# B&R Automation Studio project Panasonic_LinkaKapacitorov_A2021040 (part 4)

#### Main.st - Init, cyclic, exit code
```iecst
PROGRAM _INIT
	(* Insert code here *)

END_PROGRAM

PROGRAM _CYCLIC

	//Volanie podprogramov//
	OvlCentrovacky;
	OvlCitackyRFID;
	OvlTlaciarne;

	//Volanie funkcie SequenceControl//
	SequenceControl(SC:= SC_StoperEtiketovania);

	//Volanie funkčného bloku komunikácie Panasonic//
	KOM_Panasonic();

	//Reset sekcie //
	IF StoperEtiketovania.Reset THEN
		SC_StoperEtiketovania.Step:= 0;
		StoperEtiketovania.Reset:= FALSE;
	ELSIF NOT Safety.STAV.ZonaCS_AKTIVNA THEN
		SC_StoperEtiketovania.Step:= 0;
	END_IF

	//Status Tlačiareň zaaretovaná//
	StoperEtiketovania.STAV.TlaciarenZaaretovana:= StoperEtiketovania.IN.SuflikTlaciarne_LS_IS23 AND StoperEtiketovania.IN.SuflikTlaciarne_PS_IS22;

	//Zrušenie príznaku prebieha vyvezenie paletky//
	IF StoperEtiketovania.STAV.PrebiehaVyvazaniePaletky AND StoperDopravNG.IN.Stoper_PritomnostPaletky_IS15 THEN
		StoperEtiketovania.STAV.PrebiehaVyvazaniePaletky:= FALSE;
	END_IF

	//Označenie paletky NG pri otvoreni dverí//
	IF NOT Safety.STAV.ZamkyBunky_AKTIVNE AND RFID_Hlava_2.STAV.PritomnostCipu AND RFID_Hlava_2.PAR.PrecitaneCisloPaletky <> '' THEN
		i:=  STRING_TO_USINT(RFID_Hlava_2.PAR.PrecitaneCisloPaletky);
		IF NOT Paletka[i].StavKomunikacie_DONE THEN
			Paletka[i].StavPaletky:= 'NG';
		END_IF
	END_IF

	CASE SC_StoperEtiketovania.Step OF

		0:
			SC_StoperEtiketovania.StepName:='0 - Nulovanie';
			StoperEtiketovania.Automat:= FALSE;
			StoperEtiketovania.KoniecCyklu:= FALSE;
			StoperEtiketovania.Manual:= FALSE;
			StoperEtiketovania.STAV.PoINIT:= FALSE;
			StoperEtiketovania.OUT.StoperZASUN_YV007:= FALSE;
			SC_OvlCentrovacky.Step:= 0;
			Robot.KOM_OUT.PresunDoPozicieOdobratiaEtikety:= FALSE;
			Robot.KOM_OUT.PresunDoMutingPozicie:= FALSE;
			Robot.KOM_OUT.PresunDoPoziceKontrolyEtikety:= FALSE;
			Robot.KOM_OUT.PresunDoPoziceKontrEtiketyPriamo:= FALSE;
			Robot.KOM_OUT.PresunDoPozicieKontrolyIntStitku:= FALSE;
			Robot.KOM_OUT.NalepEtiketu:= FALSE;
			Robot.KOM_OUT.CitanieStitkuUkoncene:= FALSE;
			StoperEtiketovania.OUT.Tlaciaren_VytlacEtiketu:= FALSE;
			StoperEtiketovania.OUT.Tlaciaren_VytlacZnovaEtiketu:= FALSE;
			Kamera.STAV.Results_READY:= FALSE;
			Kamera.CMD.Triger:= FALSE;
			StoperEtiketovania.STAV.PrebiehaVyvazaniePaletky:= FALSE;
			StoperEtiketovania.RR_VytlacEtiketu:= FALSE;
			Vizu.ZobrazHlasenie_ZaaretujTlaciaren:= 1;
			Vizu.ZobrazHlas_ZatvorSerDvereTlac:= 1;
			Vizu.ZobrazHlasenie_TlaciarenOffline:= 1;
			StoperDopravNG.OUT.NatlakujTlmicPaletky_YV008:= FALSE;
			NacitanieKorekcii_DONE:= FALSE;
			StoperEtiketovania.STAV.Etiketovanie_BUSY:= FALSE;
			StoperEtiketovania_Statistika.IN.START_MeraniaCasu:= FALSE;
			KOM_Panasonic.Server_IN.DataForServer_READY:= FALSE;
			KOM_Panasonic.Server_IN.VytlacEtiketu_RucnyRezim:= FALSE;
			KOM_Panasonic.Server_IN.ProcessResult:= FALSE;
			KOM_Panasonic.Server_IN.Blowing_Error:= FALSE;
			KOM_Panasonic.Server_IN.DMcode_Reading_Error:= FALSE;
			KOM_Panasonic.Server_IN.QRcode_Reading_Error:= FALSE;
			KOM_Panasonic.Server_IN.RFID_Reading_Error:= FALSE;
			KOM_Panasonic.Server_IN.Text_Reading_Error:= FALSE;
			KOM_Panasonic.Server_IN.CommandNumber:= 0;
			KOM_Panasonic.Server_IN.RezimBezTlaceEtikety:= FALSE;
			StoperEtiketovania.STAV.Warning:= FALSE;

			IF Safety.STAV.ZonaCS_AKTIVNA AND Safety.STAV.ZonaBunky_AKTIVNA AND Linka.IN.TlakVzduchu_OK_S2 AND NOT NastalaPorucha AND Linka.STAV.Hardware_OK THEN
				SC_StoperEtiketovania.ResetStep:= TRUE;
				SC_StoperEtiketovania.Step:= 1;
			END_IF

		1:
			SC_StoperEtiketovania.StepName:='1 - Cakam na spustenie vyroby';
			StoperEtiketovania.KoniecCyklu:= FALSE;
			IF StoperEtiketovania.Automat THEN
				SC_StoperEtiketovania.Step:= 2;
			ELSIF StoperEtiketovania.Manual THEN
				SC_StoperEtiketovania.Step:= 700;
			END_IF

			//********************************************************Inicializácia****************************************************************************//

		2:
			SC_StoperEtiketovania.StepName:='2 - Inicializacia - cakam na spustenie inicializacie';
			SC_StoperEtiketovania.IdleTime.PT:= T#4s;
			SC_StoperEtiketovania.AlarmTime.PT:= T#5s;

			IF DopravBunky.STAV.PoINIT AND Robot.STAV.PoINIT THEN
				SC_StoperEtiketovania.ResetStep:= TRUE;
				SC_StoperEtiketovania.Step:= 10;
			END_IF

		10:
			SC_StoperEtiketovania.StepName:='10 - Inicializacia - zasunutie centrovacky';
			SC_StoperEtiketovania.IdleTime.PT:= T#4s;
			SC_StoperEtiketovania.AlarmTime.PT:= T#5s;

			IF NOT SC_StoperEtiketovania.Switch1 THEN
				Centrovacku_ZASUN:= TRUE;
				SC_StoperEtiketovania.Switch1:= TRUE;
			END_IF

			IF StoperEtiketovania.IN.Centrovanie_SpodnaPoloha_IS17 THEN
				SC_StoperEtiketovania.ResetStep:= TRUE;
				SC_StoperEtiketovania.Step:= 13;
			END_IF

		13:
			SC_StoperEtiketovania.StepName:='13 - Inicializacia - hladanie paletky';
			SC_StoperEtiketovania.IdleTime.PT:= T#5s;
			SC_StoperEtiketovania.AlarmTime.PT:= T#5s;
			SC_StoperEtiketovania.IdleTime.IN:= TRUE;

			IF StoperEtiketovania.IN.PritomnostPaletky_IS16 THEN
				StoperEtiketovania.STAV.PoINIT:= TRUE;
				SC_StoperEtiketovania.ResetStep:= TRUE;
				SC_StoperEtiketovania.Step:= 100;
			ELSIF SC_StoperEtiketovania.IdleTime.Q THEN
				StoperEtiketovania.STAV.PoINIT:= TRUE;
				SC_StoperEtiketovania.ResetStep:= TRUE;
				SC_StoperEtiketovania.Step:= 100;
			END_IF

			//********************************************************Automatický režim****************************************************************************//
		100:
			SC_StoperEtiketovania.StepName:='100 - Automaticky Rezim - cakam na príchod paletky na stoper';
			SC_StoperEtiketovania.IdleTime.PT:= T#200ms;
			SC_StoperEtiketovania.AlarmTime.PT:= T#5s;

			IF Linka.Rezim_BezTlaceEtikety THEN
				KOM_Panasonic.Server_IN.RezimBezTlaceEtikety:= TRUE;
			ELSE
				KOM_Panasonic.Server_IN.RezimBezTlaceEtikety:= FALSE;
			END_IF

			SC_StoperEtiketovania.IdleTime.IN:= StoperEtiketovania.IN.PritomnostPaletky_IS16;

			IF StoperEtiketovania.KoniecCyklu THEN
				SC_StoperEtiketovania.ResetStep:= TRUE;
				SC_StoperEtiketovania.Step:= 0;
			ELSIF SC_StoperEtiketovania.IdleTime.Q THEN
				StoperEtiketovania_Statistika.IN.START_MeraniaCasu:= TRUE;
				StoperEtiketovania_Statistika.IN.ZAPIS_MeraniaCasu:= TRUE;
				SC_StoperEtiketovania.ResetStep:= TRUE;
				SC_StoperEtiketovania.Step:= 103;
			END_IF

		103:
			SC_StoperEtiketovania.StepName:='103 - Automaticky Rezim - citam cislo paletky';
			SC_StoperEtiketovania.IdleTime.PT:= T#0ms;
			SC_StoperEtiketovania.AlarmTime.PT:= T#10s;

			SC_StoperEtiketovania.IdleTime.IN:= RFID_Hlava_2.STAV.PritomnostCipu;

			IF SC_StoperEtiketovania.IdleTime.Q THEN
				IF RFID_Hlava_2.PAR.PrecitaneCisloPaletky <> '' THEN
					i:=  STRING_TO_USINT(RFID_Hlava_2.PAR.PrecitaneCisloPaletky);
					IF Linka.Rezim_Priechodny THEN
						SC_StoperEtiketovania.ResetStep:= TRUE;
						SC_StoperEtiketovania.Step:= 240;
					ELSE
						SC_StoperEtiketovania.ResetStep:= TRUE;
						SC_StoperEtiketovania.Step:= 105;
					END_IF
				ELSE
					Alarmy[61]:= TRUE;
					PoruchaBunky:= TRUE;
					SC_StoperEtiketovania.ResetStep:= TRUE;
					SC_StoperEtiketovania.Step:= 0;
				END_IF
			END_IF

		105:
			SC_StoperEtiketovania.StepName:='108 - Automaticky Rezim - nacitanie offsetov pozicie lepenia zakaznickej etikety a cisla programu pre robot';
			SC_StoperEtiketovania.IdleTime.PT:= T#200ms;
			SC_StoperEtiketovania.AlarmTime.PT:= T#10s;

			OffsetRobota_NazovModelu:= Paletka[i].NazovModelu;
			Robot.KOM_OUT.CisloProduktu:= Paletka[i].Robot_CisloProgramu;
			IF Kamera.STAV.AktualneCisloProgramu <> Paletka[i].Kamera_CisloProgramu_QRkod THEN
				Kamera.PAR.ZadaneCisloProgramu:= Paletka[i].Kamera_CisloProgramu_QRkod;
			END_IF

			IF NOT SC_StoperEtiketovania.Switch1 THEN
				NacitajKorekcieRobota:= TRUE;
				SC_StoperEtiketovania.Switch1:= TRUE;
			END_IF

			IF NacitanieKorekcii_DONE THEN
				NacitanieKorekcii_DONE:= FALSE;
				IF Linka.PAR.Zvolena_PozLepenia_OffsetX <> 0 THEN
					IF Linka.PAR.Zvolena_PozLepenia_OffsetX > 0 THEN
						Robot.KOM_OUT.LepenieStitku_OffsetX:= REAL_TO_USINT(Linka.PAR.Zvolena_PozLepenia_OffsetX * 10);
						Robot.KOM_OUT.LepenieStitku_ZnamienkoOffsetX:= FALSE;
					ELSIF Linka.PAR.Zvolena_PozLepenia_OffsetX < 0 THEN
						Robot.KOM_OUT.LepenieStitku_OffsetX:= REAL_TO_USINT(ABS(Linka.PAR.Zvolena_PozLepenia_OffsetX) * 10);
						Robot.KOM_OUT.LepenieStitku_ZnamienkoOffsetX:= TRUE;
					END_IF
				ELSE
					Robot.KOM_OUT.LepenieStitku_OffsetX:= 0;
					Robot.KOM_OUT.LepenieStitku_ZnamienkoOffsetX:= FALSE;
				END_IF
				IF Linka.PAR.Zvolena_PozLepenia_OffsetY <> 0 THEN
					IF Linka.PAR.Zvolena_PozLepenia_OffsetY > 0 THEN
						Robot.KOM_OUT.LepenieStitku_OffsetY:= REAL_TO_USINT(Linka.PAR.Zvolena_PozLepenia_OffsetY * 10);
						Robot.KOM_OUT.LepenieStitku_ZnamienkoOffsetY:= FALSE;
					ELSIF Linka.PAR.Zvolena_PozLepenia_OffsetY < 0 THEN
						Robot.KOM_OUT.LepenieStitku_OffsetY:= REAL_TO_USINT(ABS(Linka.PAR.Zvolena_PozLepenia_OffsetY) * 10);
						Robot.KOM_OUT.LepenieStitku_ZnamienkoOffsetY:= TRUE;
					END_IF
				ELSE
					Robot.KOM_OUT.LepenieStitku_OffsetY:= 0;
					Robot.KOM_OUT.LepenieStitku_ZnamienkoOffsetY:= FALSE;
				END_IF
				IF Linka.PAR.Zvolena_PozLepenia_OffsetZ <> 0 THEN
					IF Linka.PAR.Zvolena_PozLepenia_OffsetZ > 0 THEN
						Robot.KOM_OUT.LepenieStitku_OffsetZ:= REAL_TO_USINT(Linka.PAR.Zvolena_PozLepenia_OffsetZ * 10);
						Robot.KOM_OUT.LepenieStitku_ZnamienkoOffsetZ:= FALSE;
					ELSIF Linka.PAR.Zvolena_PozLepenia_OffsetZ < 0 THEN
						Robot.KOM_OUT.LepenieStitku_OffsetZ:= REAL_TO_USINT(ABS(Linka.PAR.Zvolena_PozLepenia_OffsetZ) * 10);
						Robot.KOM_OUT.LepenieStitku_ZnamienkoOffsetZ:= TRUE;
					END_IF
				ELSE
					Robot.KOM_OUT.LepenieStitku_OffsetZ:= 0;
					Robot.KOM_OUT.LepenieStitku_ZnamienkoOffsetZ:= FALSE;
				END_IF
				SC_StoperEtiketovania.ResetStep:= TRUE;
				SC_StoperEtiketovania.Step:= 110;
			END_IF

		110:
			SC_StoperEtiketovania.StepName:='110 - Automaticky Rezim - zacentrovanie paletky';
			SC_StoperEtiketovania.IdleTime.PT:= T#200ms;
			SC_StoperEtiketovania.AlarmTime.PT:= T#5s;

			IF NOT SC_StoperEtiketovania.Switch1 THEN
				Centrovacku_VYSUN:= TRUE;
				SC_StoperEtiketovania.Switch1:= TRUE;
			END_IF

			IF StoperEtiketovania.IN.Centrovanie_HornaPoloha_IS18 AND NOT StoperDopravNG.STAV.DopravnikNG_BUSY THEN
				IF Linka.Rezim_BezKomunikacie THEN
					SC_StoperEtiketovania.ResetStep:= TRUE;
					SC_StoperEtiketovania.Step:= 115;
				ELSE
					SC_StoperEtiketovania.ResetStep:= TRUE;
					SC_StoperEtiketovania.Step:= 113;
				END_IF
			END_IF

		113:
			SC_StoperEtiketovania.StepName:='113 - Automaticky Rezim - kontrola stavu komunikacie a paletky';
			SC_StoperEtiketovania.IdleTime.PT:= T#200ms;
			SC_StoperEtiketovania.AlarmTime.PT:= T#5s;

			IF Paletka[i].StavKomunikacie_DONE THEN
				SC_StoperEtiketovania.ResetStep:= TRUE;
				SC_StoperEtiketovania.Step:= 240;
			ELSIF Paletka[i].StavPaletky = 'PR' THEN	//Priechodný režim
				SC_StoperEtiketovania.ResetStep:= TRUE;
				SC_StoperEtiketovania.Step:= 240;
			ELSIF Paletka[i].StavPaletky = 'NG' AND KOM_Panasonic.Server_OUT.LastCommandNumber = 0 THEN
				SC_StoperEtiketovania.ResetStep:= TRUE;
				SC_StoperEtiketovania.Step:= 240;
			ELSIF Paletka[i].StavPaletky = 'OK' AND KOM_Panasonic.Server_OUT.LastCommandNumber = 0 THEN  //Začiatok
				SC_StoperEtiketovania.ResetStep:= TRUE;
				SC_StoperEtiketovania.Step:= 115;
			ELSIF Paletka[i].StavPaletky = 'OK' AND KOM_Panasonic.Server_OUT.LastCommandNumber = 10 THEN //Načítanie internej etikety
				IF NOT StoperDopravNG.STAV.DopravnikNG_BUSY THEN
					StoperEtiketovania.STAV.Etiketovanie_BUSY:= TRUE;
					SC_StoperEtiketovania.ResetStep:= TRUE;
					SC_StoperEtiketovania.Step:= 140;
				END_IF
			ELSIF Paletka[i].StavPaletky = 'OK' AND KOM_Panasonic.Server_OUT.LastCommandNumber = 20 THEN //Vytlačenie štítku z tlačiarne
				IF NOT StoperDopravNG.STAV.DopravnikNG_BUSY THEN
					StoperEtiketovania.STAV.Etiketovanie_BUSY:= TRUE;
					SC_StoperEtiketovania.ResetStep:= TRUE;
					SC_StoperEtiketovania.Step:= 140;
				END_IF
			ELSIF Paletka[i].StavPaletky = 'OK' AND KOM_Panasonic.Server_OUT.LastCommandNumber = 30 THEN //Nalepenie štítku
				IF NOT StoperDopravNG.STAV.DopravnikNG_BUSY THEN
					StoperEtiketovania.STAV.Etiketovanie_BUSY:= TRUE;
					SC_StoperEtiketovania.ResetStep:= TRUE;
					SC_StoperEtiketovania.Step:= 180;
				END_IF
			ELSIF Paletka[i].StavPaletky = 'OK' AND KOM_Panasonic.Server_OUT.LastCommandNumber = 40 THEN //Načítanie zákaznickej etikety
				IF NOT StoperDopravNG.STAV.DopravnikNG_BUSY THEN
					StoperEtiketovania.STAV.Etiketovanie_BUSY:= TRUE;
					SC_StoperEtiketovania.ResetStep:= TRUE;
					SC_StoperEtiketovania.Step:= 180;
				END_IF
			ELSIF Paletka[i].StavPaletky = 'OK' AND KOM_Panasonic.Server_OUT.LastCommandNumber = 50 THEN //Komunikacia zo serverom ukončená
				SC_StoperEtiketovania.ResetStep:= TRUE;
				SC_StoperEtiketovania.Step:= 240;
			END_IF

		115:
			SC_StoperEtiketovania.StepName:='115 - Automaticky Rezim - presun robota na poziciu precitania interneho stitku';
			SC_StoperEtiketovania.IdleTime.PT:= T#200ms;
			SC_StoperEtiketovania.AlarmTime.PT:= T#5s;

			IF NOT StoperDopravNG.STAV.DopravnikNG_BUSY AND NOT SC_StoperEtiketovania.Switch1 THEN
				Robot.KOM_OUT.CisloProduktu:= Paletka[i].Robot_CisloProgramu;
				StoperEtiketovania.STAV.Etiketovanie_BUSY:= TRUE;
				Robot.KOM_OUT.PresunDoPozicieKontrolyIntStitku:= TRUE;
				SC_StoperEtiketovania.Switch1:= TRUE;
			END_IF

			IF Robot.KOM_IN.Stav_RobotCinnostUkoncena THEN
				Robot.KOM_OUT.PresunDoPozicieKontrolyIntStitku:= FALSE;
				SC_StoperEtiketovania.ResetStep:= TRUE;
				SC_StoperEtiketovania.Step:= 118;
			END_IF

		118:
			SC_StoperEtiketovania.StepName:='118 - Automaticky Rezim - cakam na zrusenie signalu cinnost robota ukoncena';
			SC_StoperEtiketovania.IdleTime.PT:= T#200ms;
			SC_StoperEtiketovania.AlarmTime.PT:= T#5s;

			Kamera.STAV.Results_READY:= FALSE;

			IF NOT Robot.KOM_IN.Stav_RobotCinnostUkoncena AND (Kamera.PAR.ZadaneCisloProgramu = Kamera.STAV.AktualneCisloProgramu) AND NOT Kamera.STAV.Results_READY THEN
				Kamera.STAV.Old_Hodnota_RUN_Counter:= Kamera.STAV.RUN_Counter;
				SC_StoperEtiketovania.ResetStep:= TRUE;
				SC_StoperEtiketovania.Step:= 120;
			END_IF

		120:
			SC_StoperEtiketovania.StepName:='120 - Automaticky Rezim - nacitanie interného stitku';
			SC_StoperEtiketovania.IdleTime.PT:= T#5s;
			SC_StoperEtiketovania.AlarmTime.PT:= T#5s;

			IF NOT SC_StoperEtiketovania.Switch1 AND NOT Kamera.STAV.Results_READY AND Kamera.STAV.READY THEN
				Kamera.CMD.Triger:= TRUE;
				SC_StoperEtiketovania.IdleTime.IN:= TRUE;
				SC_StoperEtiketovania.Switch1:= TRUE;
			END_IF

			IF NOT Kamera.STAV.READY THEN
				Alarmy[75]:= TRUE;
				PoruchaBunky:= TRUE;
				SC_StoperEtiketovania.ResetStep:= TRUE;
				SC_StoperEtiketovania.Step:= 0;
			ELSIF NOT Kamera.CMD.Triger AND Kamera.STAV.Results_READY THEN
				Kamera.STAV.Results_READY:= FALSE;
			ELSIF Kamera.CMD.Triger AND Kamera.STAV.Results_READY AND (Kamera.STAV.Old_Hodnota_RUN_Counter <> Kamera.STAV.RUN_Counter) THEN
				PocetOpatovnychTrigrov:= 0;
				Kamera.STAV.Results_READY:= FALSE;
				Kamera.CMD.Triger:= FALSE;
				SC_StoperEtiketovania.ResetStep:= TRUE;
				SC_StoperEtiketovania.Step:= 122;
			ELSIF SC_StoperEtiketovania.IdleTime.Q AND NOT Kamera.STAV.Results_READY THEN
				SC_StoperEtiketovania.ResetStep:= TRUE;
				SC_StoperEtiketovania.Step:= 121;
			END_IF

		121:
			SC_StoperEtiketovania.StepName:='121 - Automaticky Rezim - cakam na opatovny triger kamery';
			SC_StoperEtiketovania.IdleTime.PT:= T#2s;
			SC_StoperEtiketovania.AlarmTime.PT:= T#5s;

			Kamera.STAV.Results_READY:= FALSE;
			Kamera.CMD.Triger:= FALSE;
			Kamera.STAV.Old_Hodnota_RUN_Counter:= Kamera.STAV.RUN_Counter;
			SC_StoperEtiketovania.IdleTime.IN:= TRUE;

			IF SC_StoperEtiketovania.IdleTime.Q AND PocetOpatovnychTrigrov <= 3 THEN
				PocetOpatovnychTrigrov:= PocetOpatovnychTrigrov + 1;
				SC_StoperEtiketovania.ResetStep:= TRUE;
				SC_StoperEtiketovania.Step:= 120;
			ELSIF SC_StoperEtiketovania.IdleTime.Q AND PocetOpatovnychTrigrov > 3 THEN
				Alarmy[75]:= TRUE;
				PoruchaBunky:= TRUE;
				SC_StoperEtiketovania.ResetStep:= TRUE;
				SC_StoperEtiketovania.Step:= 0;
			END_IF

		122:
			SC_StoperEtiketovania.StepName:='122 - Automaticky Rezim - odsunutie robota po precitani interneho stitku';
			SC_StoperEtiketovania.IdleTime.PT:= T#200ms;
			SC_StoperEtiketovania.AlarmTime.PT:= T#5s;

			IF NOT SC_StoperEtiketovania.Switch1 THEN
				Robot.KOM_OUT.CitanieStitkuUkoncene:= TRUE;
				SC_StoperEtiketovania.Switch1:= TRUE;
			END_IF

			IF Robot.KOM_IN.Stav_RobotCinnostUkoncena THEN
				Robot.KOM_OUT.CitanieStitkuUkoncene:= FALSE;
				SC_StoperEtiketovania.ResetStep:= TRUE;
				SC_StoperEtiketovania.Step:= 123;
			END_IF

		123:
			SC_StoperEtiketovania.StepName:='123 - Automaticky Rezim - cakam na zrusenie signalu cinnost robota ukoncena';
			SC_StoperEtiketovania.IdleTime.PT:= T#200ms;
			SC_StoperEtiketovania.AlarmTime.PT:= T#5s;

			IF NOT Robot.KOM_IN.Stav_RobotCinnostUkoncena THEN
				SC_StoperEtiketovania.ResetStep:= TRUE;
				SC_StoperEtiketovania.Step:= 125;
			END_IF

		125:
			SC_StoperEtiketovania.StepName:='125 - Automaticky Rezim - kontrola kamerovych vysledkov citania interneho QR kodu';
			SC_StoperEtiketovania.IdleTime.PT:= T#200ms;
			SC_StoperEtiketovania.AlarmTime.PT:= T#5s;

			IF Kamera.RESULT.InternaEtiketa_QRkod_OK AND Kamera.RESULT.InternaEtiketa_ZnakyQRkodu <> 'Error' THEN
				Paletka[i].StavCitania_InternehoQRkodu:= 'OK';
				Paletka[i].InternySerialNumber:= Kamera.RESULT.InternaEtiketa_ZnakyQRkodu;
				IF Linka.Rezim_BezKomunikacie THEN
					SC_StoperEtiketovania.ResetStep:= TRUE;
					SC_StoperEtiketovania.Step:= 145;
				ELSE
					SC_StoperEtiketovania.ResetStep:= TRUE;
					SC_StoperEtiketovania.Step:= 133;
				END_IF
			ELSIF NOT Kamera.RESULT.InternaEtiketa_QRkod_OK THEN
				Paletka[i].StavCitania_InternehoQRkodu:= 'NG';
				Paletka[i].StavPaletky:= 'NG';
				Paletka[i].ReturnProcessName:= 'Neprecitany interny QR kod';
				SC_StoperEtiketovania.ResetStep:= TRUE;
				SC_StoperEtiketovania.Step:= 230;
			END_IF

		133:
			SC_StoperEtiketovania.StepName:='133 - Automaticky Rezim - odoslanie serioveho cisla internej etikety, cisla paletky a stavu cistenia na server Panasonic';
			SC_StoperEtiketovania.IdleTime.PT:= T#100ms;
			SC_StoperEtiketovania.AlarmTime.PT:= T#5s;

			KOM_Panasonic.Server_IN.NazovPaletky_RFID:= Paletka[i].NazovPaletky;
			KOM_Panasonic.Server_IN.SerialNumber_InternaEtiketa:= Paletka[i].InternySerialNumber;
			KOM_Panasonic.Server_IN.Cislo_LOTU:= Paletka[i].CisloLOT;

			IF Kamera.STAV.AktualneCisloProgramu <> Paletka[i].Kamera_CisloProgramu_DMkod THEN
				Kamera.PAR.ZadaneCisloProgramu:= Paletka[i].Kamera_CisloProgramu_DMkod;
			END_IF

			IF NOT KOM_Panasonic.Server_OUT.DataForPLC_READY THEN
				IF Paletka[i].StavCistenia = 'OK' THEN
					KOM_Panasonic.Server_IN.CommandNumber:= 10;
					KOM_Panasonic.Server_IN.ProcessResult:= TRUE;
					KOM_Panasonic.Server_IN.DataForServer_READY:= TRUE;
					SC_StoperEtiketovania.ResetStep:= TRUE;
					SC_StoperEtiketovania.Step:= 135;
				ELSIF Paletka[i].StavCistenia = 'NG' THEN
					KOM_Panasonic.Server_IN.CommandNumber:= 10;
					KOM_Panasonic.Server_IN.ProcessResult:= FALSE;
					KOM_Panasonic.Server_IN.DataForServer_READY:= TRUE;
					SC_StoperEtiketovania.ResetStep:= TRUE;
					SC_StoperEtiketovania.Step:= 135;
				END_IF
			END_IF

		135:
			SC_StoperEtiketovania.StepName:='135 - Automaticky Rezim - cakam na odpoved servera Panasonic';
			SC_StoperEtiketovania.IdleTime.PT:= T#100ms;
			SC_StoperEtiketovania.AlarmTime.PT:= T#5s;

			IF KOM_Panasonic.Server_OUT.DataForPLC_READY AND KOM_Panasonic.Server_OUT.LastCommandNumber = 10 THEN
				IF KOM_Panasonic.Server_OUT.ContinueToNextProcess THEN
					Paletka[i].ZakaznickeCislo:= KOM_Panasonic.Server_OUT.SerialNumber_ZakaznickaEtiketa;
					KOM_Panasonic.Server_IN.CommandNumber:= 0;
					KOM_Panasonic.Server_IN.DataForServer_READY:= FALSE;
					IF Linka.Rezim_BezTlaceEtikety THEN
						SC_StoperEtiketovania.ResetStep:= TRUE;
						SC_StoperEtiketovania.Step:= 190;
					ELSE
						SC_StoperEtiketovania.ResetStep:= TRUE;
						SC_StoperEtiketovania.Step:= 140;
					END_IF
				ELSIF NOT KOM_Panasonic.Server_OUT.ContinueToNextProcess THEN
					Paletka[i].ReturnProcessName:= KOM_Panasonic.Server_OUT.ReturnProcessName;
					Paletka[i].StavPaletky:= 'NG';
					KOM_Panasonic.Server_IN.CommandNumber:= 0;
					KOM_Panasonic.Server_IN.DataForServer_READY:= FALSE;
					SC_StoperEtiketovania.ResetStep:= TRUE;
					SC_StoperEtiketovania.Step:= 230;
				END_IF
			END_IF

		140:
			SC_StoperEtiketovania.StepName:='140 - Automaticky Rezim - odoslanie poziadavky na vytlacenie etikety na server Panasonic';
			SC_StoperEtiketovania.IdleTime.PT:= T#200ms;
			SC_StoperEtiketovania.AlarmTime.PT:= T#5s;

			KOM_Panasonic.Server_IN.NazovPaletky_RFID:= Paletka[i].NazovPaletky;
			KOM_Panasonic.Server_IN.SerialNumber_InternaEtiketa:= Paletka[i].InternySerialNumber;
			KOM_Panasonic.Server_IN.Cislo_LOTU:= Paletka[i].CisloLOT;

			IF NOT KOM_Panasonic.Server_OUT.DataForPLC_READY THEN
				KOM_Panasonic.Server_IN.CommandNumber:= 20;
				KOM_Panasonic.Server_IN.ProcessResult:= TRUE;
				KOM_Panasonic.Server_IN.DataForServer_READY:= TRUE;
				SC_StoperEtiketovania.ResetStep:= TRUE;
				SC_StoperEtiketovania.Step:= 145;
			END_IF

		145:
			SC_StoperEtiketovania.StepName:='145 - Automaticky Rezim - presun robota na poziciu odobratia etikety z tlaciarne';
			SC_StoperEtiketovania.IdleTime.PT:= T#200ms;
			SC_StoperEtiketovania.AlarmTime.PT:= T#5s;

			IF Kamera.STAV.AktualneCisloProgramu <> Paletka[i].Kamera_CisloProgramu_DMkod THEN
				Kamera.PAR.ZadaneCisloProgramu:= Paletka[i].Kamera_CisloProgramu_DMkod;
			END_IF

			IF StoperEtiketovania.STAV.TlaciarenZaaretovana AND NOT StoperEtiketovania.IN.Tlaciaren_Offline AND NOT SC_StoperEtiketovania.Switch1 THEN
				Robot.KOM_OUT.PresunDoPozicieOdobratiaEtikety:= TRUE;
				IF Linka.Rezim_BezKomunikacie THEN
					StoperEtiketovania.OUT.Tlaciaren_VytlacEtiketu:= TRUE;
				END_IF
				SC_StoperEtiketovania.Switch1:= TRUE;
			END_IF

			IF Robot.KOM_IN.Stav_RobotCinnostUkoncena THEN
				Robot.KOM_OUT.PresunDoPozicieOdobratiaEtikety:= FALSE;
				SC_StoperEtiketovania.ResetStep:= TRUE;
				SC_StoperEtiketovania.Step:= 148;
			END_IF

		148:
			SC_StoperEtiketovania.StepName:='148 - Automaticky Rezim - cakam na zrusenie signalu cinnost robota ukoncena';
			SC_StoperEtiketovania.IdleTime.PT:= T#200ms;
			SC_StoperEtiketovania.AlarmTime.PT:= T#5s;

			IF NOT Robot.KOM_IN.Stav_RobotCinnostUkoncena THEN
				IF Linka.Rezim_BezKomunikacie THEN
					SC_StoperEtiketovania.ResetStep:= TRUE;
					SC_StoperEtiketovania.Step:= 155;
				ELSE
					SC_StoperEtiketovania.ResetStep:= TRUE;
					SC_StoperEtiketovania.Step:= 150;
				END_IF
			END_IF

		150:
			SC_StoperEtiketovania.StepName:='150 - Automaticky Rezim - cakam na odpoved servera Panasonic';
			SC_StoperEtiketovania.IdleTime.PT:= T#200ms;
			SC_StoperEtiketovania.AlarmTime.PT:= T#5s;

			IF KOM_Panasonic.Server_OUT.DataForPLC_READY AND KOM_Panasonic.Server_OUT.LastCommandNumber = 20 THEN
				IF KOM_Panasonic.Server_OUT.ContinueToNextProcess THEN
					KOM_Panasonic.Server_IN.CommandNumber:= 0;
					KOM_Panasonic.Server_IN.DataForServer_READY:= FALSE;
					SC_StoperEtiketovania.ResetStep:= TRUE;
					SC_StoperEtiketovania.Step:= 155;
				ELSIF NOT KOM_Panasonic.Server_OUT.ContinueToNextProcess THEN
					Paletka[i].ReturnProcessName:= KOM_Panasonic.Server_OUT.ReturnProcessName;
					Paletka[i].StavPaletky:= 'NG';
					KOM_Panasonic.Server_IN.CommandNumber:= 0;
					KOM_Panasonic.Server_IN.DataForServer_READY:= FALSE;
					SC_StoperEtiketovania.ResetStep:= TRUE;
					SC_StoperEtiketovania.Step:= 230;
				END_IF
			END_IF

		155:
			SC_StoperEtiketovania.StepName:='150 - Automaticky Rezim - kontrola vytlacenia etikety';
			SC_StoperEtiketovania.IdleTime.PT:= T#500ms;
			SC_StoperEtiketovania.AlarmTime.PT:= T#20s;

			SC_StoperEtiketovania.AlarmTime.IN:= TRUE;
			SC_StoperEtiketovania.IdleTime.IN:= Robot.IN.PrisatieEtikety_OK_S1;

			IF SC_StoperEtiketovania.IdleTime.Q THEN
				SC_StoperEtiketovania.ResetStep:= TRUE;
				SC_StoperEtiketovania.Step:= 160;
			ELSIF SC_StoperEtiketovania.AlarmTime.Q THEN
				Paletka[i].StavNalepeniaEtikety:= 'NG';
				IF Linka.Rezim_BezKomunikacie THEN
					SC_StoperEtiketovania.ResetStep:= TRUE;
					SC_StoperEtiketovania.Step:= 230;
				ELSE
					Alarmy[76]:= TRUE;
					PoruchaBunky:= TRUE;
					SC_StoperEtiketovania.ResetStep:= TRUE;
					SC_StoperEtiketovania.Step:= 170;
				END_IF
			END_IF

		160:
			SC_StoperEtiketovania.StepName:='160 - Automaticky Rezim - nalepenie etikety na produkt';
			SC_StoperEtiketovania.IdleTime.PT:= T#200ms;
			SC_StoperEtiketovania.AlarmTime.PT:= T#5s;

			IF NOT SC_StoperEtiketovania.Switch1 THEN
				Robot.KOM_OUT.NalepEtiketu:= TRUE;
				SC_StoperEtiketovania.Switch1:= TRUE;
			END_IF

			IF Robot.KOM_IN.Stav_RobotCinnostUkoncena THEN
				Robot.KOM_OUT.NalepEtiketu:= FALSE;
				SC_StoperEtiketovania.ResetStep:= TRUE;
				SC_StoperEtiketovania.Step:= 165;
			END_IF

		165:
			SC_StoperEtiketovania.StepName:='165 - Automaticky Rezim - cakam na zrusenie signalu cinnost robota ukoncena';
			SC_StoperEtiketovania.IdleTime.PT:= T#200ms;
			SC_StoperEtiketovania.AlarmTime.PT:= T#5s;

			IF NOT Robot.KOM_IN.Stav_RobotCinnostUkoncena THEN
				Paletka[i].StavNalepeniaEtikety:= 'OK';
				Paletka[i].NalepenieEtikety_DONE:= TRUE;
				IF Linka.Rezim_BezKomunikacie THEN
					SC_StoperEtiketovania.ResetStep:= TRUE;
					SC_StoperEtiketovania.Step:= 190;
				ELSE
					SC_StoperEtiketovania.ResetStep:= TRUE;
					SC_StoperEtiketovania.Step:= 170;
				END_IF
			END_IF

		170:
			SC_StoperEtiketovania.StepName:='170 - Automaticky Rezim - odoslanie stavu nalepenia etikety na server Panasonic';
			SC_StoperEtiketovania.IdleTime.PT:= T#200ms;
			SC_StoperEtiketovania.AlarmTime.PT:= T#5s;

			KOM_Panasonic.Server_IN.NazovPaletky_RFID:= Paletka[i].NazovPaletky;
			KOM_Panasonic.Server_IN.SerialNumber_InternaEtiketa:= Paletka[i].InternySerialNumber;
			KOM_Panasonic.Server_IN.Cislo_LOTU:= Paletka[i].CisloLOT;

			IF NOT KOM_Panasonic.Server_OUT.DataForPLC_READY (*AND STEP*) THEN
				STEP:= FALSE;
				IF Paletka[i].StavNalepeniaEtikety = 'OK' THEN
					KOM_Panasonic.Server_IN.CommandNumber:= 30;
					KOM_Panasonic.Server_IN.ProcessResult:= TRUE;
					KOM_Panasonic.Server_IN.DataForServer_READY:= TRUE;
					SC_StoperEtiketovania.ResetStep:= TRUE;
					SC_StoperEtiketovania.Step:= 173;
				ELSIF Paletka[i].StavNalepeniaEtikety = 'NG' THEN
					KOM_Panasonic.Server_IN.CommandNumber:= 30;
					KOM_Panasonic.Server_IN.ProcessResult:= FALSE;
					KOM_Panasonic.Server_IN.DataForServer_READY:= TRUE;
					SC_StoperEtiketovania.ResetStep:= TRUE;
					SC_StoperEtiketovania.Step:= 173;
				END_IF
			END_IF

		173:
			SC_StoperEtiketovania.StepName:='173 - Automaticky Rezim - cakam na odpoved servera Panasonic';
			SC_StoperEtiketovania.IdleTime.PT:= T#200ms;
			SC_StoperEtiketovania.AlarmTime.PT:= T#5s;

			IF KOM_Panasonic.Server_OUT.DataForPLC_READY AND KOM_Panasonic.Server_OUT.LastCommandNumber = 30 THEN
				IF KOM_Panasonic.Server_OUT.ContinueToNextProcess THEN
					KOM_Panasonic.Server_IN.CommandNumber:= 0;
					KOM_Panasonic.Server_IN.DataForServer_READY:= FALSE;
					Paletka[i].NalepenieEtikety_DONE:= TRUE;
					SC_StoperEtiketovania.ResetStep:= TRUE;
					SC_StoperEtiketovania.Step:= 190;
				ELSIF NOT KOM_Panasonic.Server_OUT.ContinueToNextProcess THEN
					Paletka[i].ReturnProcessName:= KOM_Panasonic.Server_OUT.ReturnProcessName;
					Paletka[i].StavPaletky:= 'NG';
					KOM_Panasonic.Server_IN.CommandNumber:= 0;
					KOM_Panasonic.Server_IN.DataForServer_READY:= FALSE;
					SC_StoperEtiketovania.ResetStep:= TRUE;
					SC_StoperEtiketovania.Step:= 230;
				END_IF
			END_IF

		180:
			SC_StoperEtiketovania.StepName:='180 - Automaticky Rezim - presun robota na poziciu kamerovej kontroly zakaznickej etikety s pozicie mutingu';
			SC_StoperEtiketovania.IdleTime.PT:= T#200ms;
			SC_StoperEtiketovania.AlarmTime.PT:= T#5s;

			IF Kamera.STAV.AktualneCisloProgramu <> Paletka[i].Kamera_CisloProgramu_DMkod THEN
				Kamera.PAR.ZadaneCisloProgramu:= Paletka[i].Kamera_CisloProgramu_DMkod;
			END_IF

			IF NOT SC_StoperEtiketovania.Switch1 THEN
				Robot.KOM_OUT.PresunDoPoziceKontrEtiketyPriamo:= TRUE;
				SC_StoperEtiketovania.Switch1:= TRUE;
			END_IF

			IF Robot.KOM_IN.Stav_RobotCinnostUkoncena THEN
				Robot.KOM_OUT.PresunDoPoziceKontrEtiketyPriamo:= FALSE;
				SC_StoperEtiketovania.ResetStep:= TRUE;
				SC_StoperEtiketovania.Step:= 195;
			END_IF

		190:
			SC_StoperEtiketovania.StepName:='190 - Automaticky Rezim - presun robota na poziciu kamerovej kontroly zakaznickej etikety';
			SC_StoperEtiketovania.IdleTime.PT:= T#200ms;
			SC_StoperEtiketovania.AlarmTime.PT:= T#5s;

			IF Kamera.STAV.AktualneCisloProgramu <> Paletka[i].Kamera_CisloProgramu_DMkod THEN
				Kamera.PAR.ZadaneCisloProgramu:= Paletka[i].Kamera_CisloProgramu_DMkod;
			END_IF

			IF NOT SC_StoperEtiketovania.Switch1 THEN
				Robot.KOM_OUT.PresunDoPoziceKontrolyEtikety:= TRUE;
				SC_StoperEtiketovania.Switch1:= TRUE;
			END_IF

			IF Robot.KOM_IN.Stav_RobotCinnostUkoncena THEN
				Robot.KOM_OUT.PresunDoPoziceKontrolyEtikety:= FALSE;
				SC_StoperEtiketovania.ResetStep:= TRUE;
				SC_StoperEtiketovania.Step:= 195;
			END_IF

		195:
			SC_StoperEtiketovania.StepName:='195 - Automaticky Rezim - cakam na zrusenie signalu cinnost robota ukoncena';
			SC_StoperEtiketovania.IdleTime.PT:= T#200ms;
			SC_StoperEtiketovania.AlarmTime.PT:= T#5s;

			Kamera.STAV.Results_READY:= FALSE;

			IF NOT Robot.KOM_IN.Stav_RobotCinnostUkoncena AND (Kamera.PAR.ZadaneCisloProgramu = Kamera.STAV.AktualneCisloProgramu) AND NOT Kamera.STAV.Results_READY THEN
				Kamera.STAV.Old_Hodnota_RUN_Counter:= Kamera.STAV.RUN_Counter;
				SC_StoperEtiketovania.ResetStep:= TRUE;
				SC_StoperEtiketovania.Step:= 200;
			END_IF

		200:
			SC_StoperEtiketovania.StepName:='200 - Automaticky Rezim - kamerova kontrola zakaznickej etikety';
			SC_StoperEtiketovania.IdleTime.PT:= T#5s;
			SC_StoperEtiketovania.AlarmTime.PT:= T#5s;

			IF NOT SC_StoperEtiketovania.Switch1 AND NOT Kamera.STAV.Results_READY AND Kamera.STAV.READY THEN
				Kamera.CMD.Triger:= TRUE;
				SC_StoperEtiketovania.IdleTime.IN:= TRUE;
				SC_StoperEtiketovania.Switch1:= TRUE;
			END_IF

			IF NOT Kamera.STAV.READY THEN
				Alarmy[75]:= TRUE;
				PoruchaBunky:= TRUE;
				SC_StoperEtiketovania.ResetStep:= TRUE;
				SC_StoperEtiketovania.Step:= 0;
			ELSIF NOT Kamera.CMD.Triger AND Kamera.STAV.Results_READY THEN
				Kamera.STAV.Results_READY:= FALSE;
			ELSIF Kamera.CMD.Triger AND Kamera.STAV.Results_READY AND (Kamera.STAV.Old_Hodnota_RUN_Counter <> Kamera.STAV.RUN_Counter) THEN
				Kamera.STAV.Results_READY:= FALSE;
				Kamera.CMD.Triger:= FALSE;
				PocetOpatovnychTrigrov:= 0;
				SC_StoperEtiketovania.ResetStep:= TRUE;
				SC_StoperEtiketovania.Step:= 205;
			ELSIF SC_StoperEtiketovania.IdleTime.Q AND NOT Kamera.STAV.Results_READY THEN
				SC_StoperEtiketovania.ResetStep:= TRUE;
				SC_StoperEtiketovania.Step:= 201;
			END_IF

		201:
			SC_StoperEtiketovania.StepName:='201 - Automaticky Rezim - cakam na opatovny triger kamery';
			SC_StoperEtiketovania.IdleTime.PT:= T#2s;
			SC_StoperEtiketovania.AlarmTime.PT:= T#5s;

			Kamera.STAV.Results_READY:= FALSE;
			Kamera.CMD.Triger:= FALSE;
			Kamera.STAV.Old_Hodnota_RUN_Counter:= Kamera.STAV.RUN_Counter;
			SC_StoperEtiketovania.IdleTime.IN:= TRUE;

			IF SC_StoperEtiketovania.IdleTime.Q AND PocetOpatovnychTrigrov <= 3 THEN
				PocetOpatovnychTrigrov:= PocetOpatovnychTrigrov + 1;
				SC_StoperEtiketovania.ResetStep:= TRUE;
				SC_StoperEtiketovania.Step:= 200;
			ELSIF SC_StoperEtiketovania.IdleTime.Q AND PocetOpatovnychTrigrov > 3 THEN
				Alarmy[75]:= TRUE;
				PoruchaBunky:= TRUE;
				SC_StoperEtiketovania.ResetStep:= TRUE;
				SC_StoperEtiketovania.Step:= 0;
			END_IF

		205:
			SC_StoperEtiketovania.StepName:='205 - Automaticky Rezim - odsunutie robota po precitani zakaznickej etikety';
			SC_StoperEtiketovania.IdleTime.PT:= T#200ms;
			SC_StoperEtiketovania.AlarmTime.PT:= T#5s;

			IF NOT SC_StoperEtiketovania.Switch1 THEN
				Robot.KOM_OUT.CitanieStitkuUkoncene:= TRUE;
				SC_StoperEtiketovania.Switch1:= TRUE;
			END_IF

			IF Robot.KOM_IN.Stav_RobotCinnostUkoncena THEN
				Robot.KOM_OUT.CitanieStitkuUkoncene:= FALSE;
				SC_StoperEtiketovania.ResetStep:= TRUE;
				SC_StoperEtiketovania.Step:= 208;
			END_IF

		208:
			SC_StoperEtiketovania.StepName:='208 - Automaticky Rezim - cakam na zrusenie signalu cinnost robota ukoncena';
			SC_StoperEtiketovania.IdleTime.PT:= T#200ms;
			SC_StoperEtiketovania.AlarmTime.PT:= T#5s;

			IF NOT Robot.KOM_IN.Stav_RobotCinnostUkoncena THEN
				Centrovacku_ZASUN:= TRUE;
				SC_StoperEtiketovania.ResetStep:= TRUE;
				SC_StoperEtiketovania.Step:= 210;
			END_IF

		210:
			SC_StoperEtiketovania.StepName:='210 - Automaticky Rezim - kontrola precitania zakaznickeho DM kodu';
			SC_StoperEtiketovania.IdleTime.PT:= T#200ms;
			SC_StoperEtiketovania.AlarmTime.PT:= T#5s;

			IF Kamera.RESULT.ZakazEtiketa_DMkod_OK AND Kamera.RESULT.ZakazEtiketa_ZnakyDMkodu <> 'Error' THEN
				Paletka[i].PrecitaneZnakyZakaznickehoDMkodu:= Kamera.RESULT.ZakazEtiketa_ZnakyDMkodu;
				IF Paletka[i].ZakaznickeCislo = Paletka[i].PrecitaneZnakyZakaznickehoDMkodu THEN
					Paletka[i].StavPorovnaniaDMkoduZoServerom:= 'OK';
					Paletka[i].StavCitania_ZakaznickehoDMkodu:= 'OK';
				ELSE
					Paletka[i].StavPorovnaniaDMkoduZoServerom:= 'NG';
					Paletka[i].StavCitania_ZakaznickehoDMkodu:= 'NG';
					Paletka[i].StavPaletky:= 'NG';
				END_IF
				SC_StoperEtiketovania.ResetStep:= TRUE;
				SC_StoperEtiketovania.Step:= 215;
			ELSIF NOT Kamera.RESULT.ZakazEtiketa_DMkod_OK THEN
				Paletka[i].StavCitania_ZakaznickehoDMkodu:= 'NG';
				Paletka[i].StavPaletky:= 'NG';
				SC_StoperEtiketovania.ResetStep:= TRUE;
				SC_StoperEtiketovania.Step:= 215;
			END_IF

		215:
			SC_StoperEtiketovania.StepName:='215 - Automaticky Rezim - kontrola pritomnosti znakov na zakaznickej etikete';
			SC_StoperEtiketovania.IdleTime.PT:= T#200ms;
			SC_StoperEtiketovania.AlarmTime.PT:= T#5s;

			IF Kamera.RESULT.ZakazEtiketa_PritomnZnakov_OK (*AND Kamera.RESULT.BielyPatern_OK*) THEN
				Paletka[i].StavKontrolyBielehoPaternu:= 'OK';
				Paletka[i].StavCitania_KontrolaZnakov:= 'OK';
				IF Linka.Rezim_BezKomunikacie THEN
					SC_StoperEtiketovania.ResetStep:= TRUE;
					SC_StoperEtiketovania.Step:= 240;
				ELSE
					SC_StoperEtiketovania.ResetStep:= TRUE;
					SC_StoperEtiketovania.Step:= 220;
				END_IF
			ELSIF NOT Kamera.RESULT.ZakazEtiketa_PritomnZnakov_OK (*OR NOT Kamera.RESULT.BielyPatern_OK*) THEN
				IF NOT Kamera.RESULT.BielyPatern_OK THEN
					Paletka[i].StavKontrolyBielehoPaternu:= 'NG';
				ELSE
					Paletka[i].StavCitania_KontrolaZnakov:= 'OK';
				END_IF
				Paletka[i].StavCitania_KontrolaZnakov:= 'NG';
				Paletka[i].StavPaletky:= 'NG';
				IF Linka.Rezim_BezKomunikacie THEN
					SC_StoperEtiketovania.ResetStep:= TRUE;
					SC_StoperEtiketovania.Step:= 230;
				ELSE
					SC_StoperEtiketovania.ResetStep:= TRUE;
					SC_StoperEtiketovania.Step:= 220;
				END_IF
			END_IF

		220:
			SC_StoperEtiketovania.StepName:='220 - Automaticky Rezim - odoslanie stavu citania DM kodu zakaznickej etikety na server Panasonic';
			SC_StoperEtiketovania.IdleTime.PT:= T#200ms;
			SC_StoperEtiketovania.AlarmTime.PT:= T#5s;

			KOM_Panasonic.Server_IN.NazovPaletky_RFID:= Paletka[i].NazovPaletky;
			KOM_Panasonic.Server_IN.SerialNumber_InternaEtiketa:= Paletka[i].InternySerialNumber;
			KOM_Panasonic.Server_IN.Cislo_LOTU:= Paletka[i].CisloLOT;

			IF NOT KOM_Panasonic.Server_OUT.DataForPLC_READY (*AND STEP*) THEN
				STEP:= FALSE;
				IF Paletka[i].StavCitania_ZakaznickehoDMkodu = 'OK' THEN
					KOM_Panasonic.Server_IN.CommandNumber:= 40;
					KOM_Panasonic.Server_IN.ProcessResult:= TRUE;
					KOM_Panasonic.Server_IN.DataForServer_READY:= TRUE;
					SC_StoperEtiketovania.ResetStep:= TRUE;
					SC_StoperEtiketovania.Step:= 223;
				ELSIF Paletka[i].StavCitania_ZakaznickehoDMkodu = 'NG' THEN
					KOM_Panasonic.Server_IN.CommandNumber:= 40;
					KOM_Panasonic.Server_IN.ProcessResult:= FALSE;
					KOM_Panasonic.Server_IN.DataForServer_READY:= TRUE;
					SC_StoperEtiketovania.ResetStep:= TRUE;
					SC_StoperEtiketovania.Step:= 223;
				END_IF
			END_IF

		223:
			SC_StoperEtiketovania.StepName:='223 - Automaticky Rezim - cakam na odpoved servera Panasonic';
			SC_StoperEtiketovania.IdleTime.PT:= T#200ms;
			SC_StoperEtiketovania.AlarmTime.PT:= T#5s;

			IF KOM_Panasonic.Server_OUT.DataForPLC_READY AND KOM_Panasonic.Server_OUT.LastCommandNumber = 40 THEN
				IF KOM_Panasonic.Server_OUT.ContinueToNextProcess THEN
					KOM_Panasonic.Server_IN.CommandNumber:= 0;
					KOM_Panasonic.Server_IN.DataForServer_READY:= FALSE;
					SC_StoperEtiketovania.ResetStep:= TRUE;
					SC_StoperEtiketovania.Step:= 225;
				ELSIF NOT KOM_Panasonic.Server_OUT.ContinueToNextProcess THEN
					Paletka[i].ReturnProcessName:= KOM_Panasonic.Server_OUT.ReturnProcessName;
					Paletka[i].StavPaletky:= 'NG';
					KOM_Panasonic.Server_IN.CommandNumber:= 0;
					KOM_Panasonic.Server_IN.DataForServer_READY:= FALSE;
					SC_StoperEtiketovania.ResetStep:= TRUE;
					SC_StoperEtiketovania.Step:= 230;
				END_IF
			END_IF

		225:
			SC_StoperEtiketovania.StepName:='225 - Automaticky Rezim - odoslanie stavu citania znakov zakaznickej etikety na server Panasonic';
			SC_StoperEtiketovania.IdleTime.PT:= T#200ms;
			SC_StoperEtiketovania.AlarmTime.PT:= T#5s;

			KOM_Panasonic.Server_IN.NazovPaletky_RFID:= Paletka[i].NazovPaletky;
			KOM_Panasonic.Server_IN.SerialNumber_InternaEtiketa:= Paletka[i].InternySerialNumber;
			KOM_Panasonic.Server_IN.Cislo_LOTU:= Paletka[i].CisloLOT;

			IF NOT KOM_Panasonic.Server_OUT.DataForPLC_READY (*AND STEP*) THEN
				STEP:= FALSE;
				IF Paletka[i].StavCitania_KontrolaZnakov = 'OK' THEN
					KOM_Panasonic.Server_IN.CommandNumber:= 50;
					KOM_Panasonic.Server_IN.ProcessResult:= TRUE;
					KOM_Panasonic.Server_IN.DataForServer_READY:= TRUE;
					SC_StoperEtiketovania.ResetStep:= TRUE;
					SC_StoperEtiketovania.Step:= 228;
				ELSIF Paletka[i].StavCitania_KontrolaZnakov = 'NG' THEN
					KOM_Panasonic.Server_IN.CommandNumber:= 50;
					KOM_Panasonic.Server_IN.ProcessResult:= FALSE;
					KOM_Panasonic.Server_IN.DataForServer_READY:= TRUE;
					SC_StoperEtiketovania.ResetStep:= TRUE;
					SC_StoperEtiketovania.Step:= 228;
				END_IF
			END_IF

		228:
			SC_StoperEtiketovania.StepName:='228 - Automaticky Rezim - cakam na odpoved servera Panasonic';
			SC_StoperEtiketovania.IdleTime.PT:= T#200ms;
			SC_StoperEtiketovania.AlarmTime.PT:= T#5s;

			IF KOM_Panasonic.Server_OUT.DataForPLC_READY AND KOM_Panasonic.Server_OUT.LastCommandNumber = 50 THEN
				IF KOM_Panasonic.Server_OUT.ContinueToNextProcess THEN
					KOM_Panasonic.Server_IN.CommandNumber:= 0;
					KOM_Panasonic.Server_IN.DataForServer_READY:= FALSE;
					SC_StoperEtiketovania.ResetStep:= TRUE;
					SC_StoperEtiketovania.Step:= 240;
				ELSIF NOT KOM_Panasonic.Server_OUT.ContinueToNextProcess THEN
					Paletka[i].ReturnProcessName:= KOM_Panasonic.Server_OUT.ReturnProcessName;
					Paletka[i].StavPaletky:= 'NG';
					KOM_Panasonic.Server_IN.CommandNumber:= 0;
					KOM_Panasonic.Server_IN.DataForServer_READY:= FALSE;
					SC_StoperEtiketovania.ResetStep:= TRUE;
					SC_StoperEtiketovania.Step:= 230;
				END_IF
			END_IF

		230:
			SC_StoperEtiketovania.StepName:='230 - Automaticky Rezim - presun robota do pozicie mutingu';
			SC_StoperEtiketovania.IdleTime.PT:= T#200ms;
			SC_StoperEtiketovania.AlarmTime.PT:= T#5s;

			Paletka[i].StavKomunikacie_DONE:= TRUE;

			IF NOT SC_StoperEtiketovania.Switch1 THEN
				Robot.KOM_OUT.PresunDoMutingPozicie:= TRUE;
				SC_StoperEtiketovania.Switch1:= TRUE;
			END_IF

			IF Robot.KOM_IN.Stav_RobotCinnostUkoncena THEN
				Robot.KOM_OUT.PresunDoMutingPozicie:= FALSE;
				SC_StoperEtiketovania.ResetStep:= TRUE;
				SC_StoperEtiketovania.Step:= 235;
			END_IF

		235:
			SC_StoperEtiketovania.StepName:='235 - Automaticky Rezim - cakam na zrusenie signalu cinnost robota ukoncena';
			SC_StoperEtiketovania.IdleTime.PT:= T#200ms;
			SC_StoperEtiketovania.AlarmTime.PT:= T#5s;

			IF NOT Robot.KOM_IN.Stav_RobotCinnostUkoncena AND Safety.STAV.MutingRobota_AKTIVNY THEN
				SC_StoperEtiketovania.ResetStep:= TRUE;
				SC_StoperEtiketovania.Step:= 240;
			END_IF

		240:
			SC_StoperEtiketovania.StepName:='240 - Automaticky Rezim - odcentrovanie paletky';
			SC_StoperEtiketovania.IdleTime.PT:= T#200ms;
			SC_StoperEtiketovania.AlarmTime.PT:= T#5s;

			IF Kamera.STAV.AktualneCisloProgramu <> Paletka[i].Kamera_CisloProgramu_QRkod THEN
				Kamera.PAR.ZadaneCisloProgramu:= Paletka[i].Kamera_CisloProgramu_QRkod;
			END_IF
			StoperEtiketovania.STAV.Etiketovanie_BUSY:= FALSE;
			Paletka[i].StavKomunikacie_DONE:= TRUE;

			IF NOT SC_StoperEtiketovania.Switch1 THEN
				Centrovacku_ZASUN:= TRUE;
				SC_StoperEtiketovania.Switch1:= TRUE;
			END_IF

			IF StoperEtiketovania.IN.Centrovanie_SpodnaPoloha_IS17 THEN
				SC_StoperEtiketovania.ResetStep:= TRUE;
				SC_StoperEtiketovania.Step:= 250;
			END_IF

		250:
			SC_StoperEtiketovania.StepName:='250 - Automaticky Rezim - cakam na vyvezenie paletky na stoper dopravnika NG';
			SC_StoperEtiketovania.IdleTime.PT:= T#500ms;
			SC_StoperEtiketovania.AlarmTime.PT:= T#5s;

			StoperEtiketovania.STAV.Warning:= Paletka[i].StavPaletky = 'NG' AND StoperDopravNG.IN.Dopravnik_PritomnostPaletky_OS4;

			IF StoperEtiketovania.KoniecCyklu THEN
				SC_StoperEtiketovania.ResetStep:= TRUE;
				SC_StoperEtiketovania.Step:= 0;
			ELSIF Paletka[i].StavPaletky = 'PR' AND SC_StoperDopravNG.Step = 100 AND StoperDopravNG.IN.Centrovanie_StrednaPoloha_IS20 AND NOT StoperDopravNG.IN.Stoper_PritomnostPaletky_IS15 AND NOT StoperDopravNG.STAV.ObsluhaPotvrdilaPaletkuNG AND NOT StoperDopravNG.STAV.DopravnikNG_BUSY THEN
				StoperEtiketovania.STAV.VyvazamPaletkuNG:= FALSE;
				StoperEtiketovania.STAV.Warning:= FALSE;
				SC_StoperEtiketovania.ResetStep:= TRUE;
				SC_StoperEtiketovania.Step:= 255;
			ELSIF Paletka[i].StavPaletky = 'OK' AND SC_StoperDopravNG.Step = 100 AND StoperDopravNG.IN.Centrovanie_StrednaPoloha_IS20 AND NOT StoperDopravNG.IN.Stoper_PritomnostPaletky_IS15 AND NOT StoperDopravNG.STAV.ObsluhaPotvrdilaPaletkuNG AND NOT StoperDopravNG.STAV.DopravnikNG_BUSY THEN
				StoperEtiketovania.STAV.VyvazamPaletkuNG:= FALSE;
				PocetVyrobenychKusov_OK:= PocetVyrobenychKusov_OK + 1;
				CelkovyPocetVyrobenychKusov:= CelkovyPocetVyrobenychKusov + 1;
				StoperEtiketovania.STAV.Warning:= FALSE;
				SC_StoperEtiketovania.ResetStep:= TRUE;
				SC_StoperEtiketovania.Step:= 255;
			ELSIF Paletka[i].StavPaletky = 'NG' AND SC_StoperDopravNG.Step = 100 AND StoperDopravNG.IN.Centrovanie_StrednaPoloha_IS20 AND NOT StoperDopravNG.IN.Stoper_PritomnostPaletky_IS15 AND (NOT StoperDopravNG.IN.Dopravnik_PritomnostPaletky_OS4 AND NOT StoperDopravNG.STAV.PaletkaNaKonciDopravnika_NG) AND NOT StoperDopravNG.STAV.DopravnikNG_BUSY THEN
				StoperEtiketovania.STAV.VyvazamPaletkuNG:= TRUE;
				StoperDopravNG.STAV.DopravnikNG_BUSY:= TRUE;
				StoperEtiketovania.STAV.AlarmTextPaletkyNG:= Paletka[i].ReturnProcessName;
				PocetVyrobenychKusov_NG:= PocetVyrobenychKusov_NG + 1;
				CelkovyPocetVyrobenychKusov:= CelkovyPocetVyrobenychKusov + 1;
				StoperEtiketovania.STAV.Warning:= FALSE;
				SC_StoperEtiketovania.ResetStep:= TRUE;
				SC_StoperEtiketovania.Step:= 255;
			END_IF

		255:
			SC_StoperEtiketovania.StepName:='255 - Automaticky Rezim - vyvazam paletku na stoper dopravnika NG';
			SC_StoperEtiketovania.IdleTime.PT:= T#4s;
			SC_StoperEtiketovania.AlarmTime.PT:= T#10s;

			IF NOT SC_StoperEtiketovania.Switch1 THEN
				StoperEtiketovania.OUT.StoperZASUN_YV007:= TRUE;
				StoperDopravNG.OUT.NatlakujTlmicPaletky_YV008:= TRUE;
				StoperEtiketovania.STAV.PrebiehaVyvazaniePaletky:= TRUE;
				SC_StoperEtiketovania.AlarmTime.IN:= TRUE;
				SC_StoperEtiketovania.Switch1:= TRUE;
			END_IF

			IF NOT StoperEtiketovania.IN.PritomnostPaletky_IS16 THEN
				StoperEtiketovania.OUT.StoperZASUN_YV007:= FALSE;
				StoperDopravNG.OUT.NatlakujTlmicPaletky_YV008:= FALSE;
			END_IF

			IF NOT Linka.Rezim_Priechodny AND NOT StoperEtiketovania.IN.PritomnostPaletky_IS16 AND NOT StoperEtiketovania.OUT.StoperZASUN_YV007 THEN
				SC_StoperEtiketovania.ResetStep:= TRUE;
				SC_StoperEtiketovania.Step:= 100;
			ELSIF Linka.Rezim_Priechodny AND NOT StoperEtiketovania.IN.PritomnostPaletky_IS16 AND NOT StoperEtiketovania.OUT.StoperZASUN_YV007 AND StoperDopravNG.IN.Stoper_PritomnostPaletky_IS15 THEN
				SC_StoperEtiketovania.ResetStep:= TRUE;
				SC_StoperEtiketovania.Step:= 100;
			END_IF

			IF SC_StoperEtiketovania.AlarmTime.Q THEN
				Alarmy[56]:= TRUE;
				PoruchaBunky:= TRUE;
				SC_StoperEtiketovania.ResetStep:= TRUE;
				SC_StoperEtiketovania.Step:= 0;
			END_IF

			//*******************************************************Manuálny režim*******************************************************************************//
		700:
			SC_StoperEtiketovania.StepName:='700 - Manualny Rezim';
			SC_StoperEtiketovania.IdleTime.PT:= T#8s;
			SC_StoperEtiketovania.AlarmTime.PT:= T#5s;

			//Vytlačenie etikety//
			IF StoperEtiketovania.RR_VytlacEtiketu THEN
				IF NOT StoperEtiketovania.IN.Tlaciaren_Offline THEN
					CasVytlaceniaEtikety.IN:= TRUE;
					KOM_Panasonic.Server_IN.SerialNumber_InternaEtiketa:= '';
					strcat(ADR(KOM_Panasonic.Server_IN.SerialNumber_InternaEtiketa),ADR(StoperEtiketovania.PAR.TypPaletky_RucneVytlacEtikety));
					strcat(ADR(KOM_Panasonic.Server_IN.SerialNumber_InternaEtiketa),ADR('00000000000000000000000000'));
					KOM_Panasonic.Server_IN.VytlacEtiketu_RucnyRezim:= TRUE;
				END_IF
				StoperEtiketovania.RR_VytlacEtiketu:= FALSE;
			END_IF

			IF CasVytlaceniaEtikety.Q THEN
				KOM_Panasonic.Server_IN.VytlacEtiketu_RucnyRezim:= FALSE;
				CasVytlaceniaEtikety.IN:= FALSE;
			END_IF

			CasVytlaceniaEtikety.PT:= T#1s;
			CasVytlaceniaEtikety();

	END_CASE

END_PROGRAM

PROGRAM _EXIT
	(* Insert code here *)

END_PROGRAM
```

#### Variables.var - Local variables
```iecst
VAR
	SC_OvlCentrovacky : SequenceControlTyp;
	Centrovacku_VYSUN : BOOL;
	Centrovacku_ZASUN : BOOL;
	i : USINT := 0;
	VstupnePoleUSINT : ARRAY[1..20] OF USINT;
	VystupnePoleStringov : ARRAY[1..20] OF STRING[80];
	h : USINT := 0;
	PocetZnakovUDINT : UDINT;
	PocetZnakovUSINT : USINT;
	g : USINT := 0;
	AktualNacitanyZnak : USINT;
	CasVytlaceniaEtikety : TON := (0);
	TextovaPremenna_1 : STRING[10] := '';
	PrvyRiadok : STRING[20] := '';
	DruhyRiadok : STRING[30] := '';
	TretiRiadok : STRING[10] := '';
	DataMetrix : STRING[30] := '';
	CisloPaletky : STRING[10] := '';
	STEP : BOOL := 0;
	PocetOpatovnychTrigrov : USINT := 0;
END_VAR
```

#### OvlCentrovacky.st
```iecst
ACTION OvlCentrovacky:

	//Volanie funkcie SequenceControl//
	SequenceControl(SC:= SC_OvlCentrovacky);

	CASE SC_OvlCentrovacky.Step OF

		0:
			SC_OvlCentrovacky.StepName:= '0 - Nulovanie';
			Centrovacku_VYSUN:= FALSE;
			Centrovacku_ZASUN:= FALSE;
			StoperEtiketovania.RR_OdcentrujPaletku:= FALSE;
			StoperEtiketovania.RR_ZacentrujPaletku:= FALSE;
			//StoperEtiketovania.OUT.Centrovanie_VYSUN_YV003:= FALSE;
			//StoperEtiketovania.OUT.Centrovanie_ZASUN_YV004:= FALSE;

			IF SC_StoperEtiketovania.Step <> 0 THEN
				SC_OvlCentrovacky.ResetStep:= TRUE;
				SC_OvlCentrovacky.Step:= 1;
			END_IF

		1:
			SC_OvlCentrovacky.StepName:= '1 - Rozhodnutie o cinnosti';
			IF Centrovacku_VYSUN THEN
				SC_OvlCentrovacky.Step:= 10;
			ELSIF Centrovacku_ZASUN THEN
				SC_OvlCentrovacky.Step:= 20;
			ELSIF StoperEtiketovania.RR_ZacentrujPaletku THEN
				SC_OvlCentrovacky.Step:= 10;
			ELSIF StoperEtiketovania.RR_OdcentrujPaletku THEN
				SC_OvlCentrovacky.Step:= 20;
			END_IF

		10:
			SC_OvlCentrovacky.StepName:= '10 - Vysunutie centrovacky';
			SC_OvlCentrovacky.IdleTime.PT:= T#3s;
			SC_OvlCentrovacky.AlarmTime.PT:= T#6s;

			IF StoperEtiketovania.Automat THEN
				SC_OvlCentrovacky.AlarmTime.IN:= TRUE;
			ELSE
				SC_OvlCentrovacky.IdleTime.IN:= TRUE;
			END_IF

			IF NOT SC_OvlCentrovacky.Switch1 THEN
				StoperEtiketovania.OUT.Centrovanie_ZASUN_YV004:= FALSE;
				StoperEtiketovania.OUT.Centrovanie_VYSUN_YV003:= TRUE;
				SC_OvlCentrovacky.Switch1:= TRUE;
			END_IF

			IF StoperEtiketovania.IN.Centrovanie_HornaPoloha_IS18 OR SC_OvlCentrovacky.IdleTime.Q THEN
				SC_OvlCentrovacky.ResetStep:= TRUE;
				SC_OvlCentrovacky.Step:= 0;
			ELSIF SC_OvlCentrovacky.AlarmTime.Q THEN
				Alarmy[53]:= TRUE;
				PoruchaBunky:= TRUE;
				SC_OvlCentrovacky.ResetStep:= TRUE;
				SC_OvlCentrovacky.Step:= 0;
			END_IF

		20:
			SC_OvlCentrovacky.StepName:= '20 - Zasunutie centrovacky';
			SC_OvlCentrovacky.IdleTime.PT:= T#3s;
			SC_OvlCentrovacky.AlarmTime.PT:= T#6s;

			IF StoperEtiketovania.Automat THEN
				SC_OvlCentrovacky.AlarmTime.IN:= TRUE;
			ELSE
				SC_OvlCentrovacky.IdleTime.IN:= TRUE;
			END_IF

			IF NOT SC_OvlCentrovacky.Switch1 THEN
				StoperEtiketovania.OUT.Centrovanie_VYSUN_YV003:= FALSE;
				StoperEtiketovania.OUT.Centrovanie_ZASUN_YV004:= TRUE;
				SC_OvlCentrovacky.Switch1:= TRUE;
			END_IF

			IF StoperEtiketovania.IN.Centrovanie_SpodnaPoloha_IS17 OR SC_OvlCentrovacky.IdleTime.Q THEN
				SC_OvlCentrovacky.ResetStep:= TRUE;
				SC_OvlCentrovacky.Step:= 0;
			ELSIF SC_OvlCentrovacky.AlarmTime.Q THEN
				Alarmy[54]:= TRUE;
				PoruchaBunky:= TRUE;
				SC_OvlCentrovacky.ResetStep:= TRUE;
				SC_OvlCentrovacky.Step:= 0;
			END_IF

	END_CASE

END_ACTION
```

#### OvlCitackyRFID.st
```iecst
ACTION OvlCitackyRFID:

//***********************************************************************Riadenie RFID hlavy 2 - Pozícia nalepovania etikety**********************************************************************//

	//Volanie funkcie SequenceControl//
	SequenceControl(SC:= SC_Hlava_2);

	//*************************Komunikácia*******************************//
	//INPUTS//
	RFID_Hlava_2.STAV.PritomnostCipu:= RFID_Hlava_2.IN.BYTE_IN[0].0;
	RFID_Hlava_2.IN.Bit_CP:= RFID_Hlava_2.IN.BYTE_IN[0].0;
	RFID_Hlava_2.IN.Bit_AA:= RFID_Hlava_2.IN.BYTE_IN[0].1;
	RFID_Hlava_2.IN.Bit_AE:= RFID_Hlava_2.IN.BYTE_IN[0].2;
	RFID_Hlava_2.IN.Bit_AF:= RFID_Hlava_2.IN.BYTE_IN[0].3;
	RFID_Hlava_2.IN.Bit_MT:= RFID_Hlava_2.IN.BYTE_IN[0].4;
	RFID_Hlava_2.IN.Bit_TO:= RFID_Hlava_2.IN.BYTE_IN[0].5;
	RFID_Hlava_2.IN.Bit_HF:= RFID_Hlava_2.IN.BYTE_IN[0].6;
	RFID_Hlava_2.IN.Bit_BB:= RFID_Hlava_2.IN.BYTE_IN[0].7;

	//OUTPUTS//
	RFID_Hlava_2.OUT.BYTE_OUT[0].0:= RFID_Hlava_2.OUT.Bit_AV;
	RFID_Hlava_2.OUT.BYTE_OUT[31].0:= RFID_Hlava_2.OUT.Bit_AV;
	RFID_Hlava_2.OUT.BYTE_OUT[0].2:= RFID_Hlava_2.OUT.Bit_GR;
	RFID_Hlava_2.OUT.BYTE_OUT[31].2:= RFID_Hlava_2.OUT.Bit_GR;
	RFID_Hlava_2.OUT.BYTE_OUT[0].5:= RFID_Hlava_2.OUT.Bit_KA;
	RFID_Hlava_2.OUT.BYTE_OUT[31].5:= RFID_Hlava_2.OUT.Bit_KA;
	RFID_Hlava_2.OUT.BYTE_OUT[0].6:= RFID_Hlava_2.OUT.Bit_TI;
	RFID_Hlava_2.OUT.BYTE_OUT[31].6:= RFID_Hlava_2.OUT.Bit_TI;

	//Prečítané znaky//
	RFID_Hlava_2.PAR.PrecitaneCisloPaletky_POLE[0]:= RFID_Hlava_2.IN.BYTE_IN[1];
	RFID_Hlava_2.PAR.PrecitaneCisloPaletky_POLE[1]:= RFID_Hlava_2.IN.BYTE_IN[2];
	RFID_Hlava_2.PAR.PrecitaneCisloPaletky_POLE[2]:= RFID_Hlava_2.IN.BYTE_IN[3];
	RFID_Hlava_2.PAR.PrecitaneCisloPaletky_POLE[3]:= RFID_Hlava_2.IN.BYTE_IN[4];
	RFID_Hlava_2.PAR.PrecitaneCisloPaletky_POLE[4]:= RFID_Hlava_2.IN.BYTE_IN[5];
	RFID_Hlava_2.PAR.PrecitaneCisloPaletky_POLE[5]:= RFID_Hlava_2.IN.BYTE_IN[6];
	RFID_Hlava_2.PAR.PrecitaneCisloPaletky_POLE[6]:= RFID_Hlava_2.IN.BYTE_IN[7];
	RFID_Hlava_2.PAR.PrecitaneCisloPaletky_POLE[7]:= RFID_Hlava_2.IN.BYTE_IN[8];
	RFID_Hlava_2.PAR.PrecitaneCisloPaletky_POLE[8]:= RFID_Hlava_2.IN.BYTE_IN[9];
	RFID_Hlava_2.PAR.PrecitaneCisloPaletky_POLE[9]:= RFID_Hlava_2.IN.BYTE_IN[10];

	brsmemcpy(ADR(RFID_Hlava_2.PAR.Precitane_Cislo_Typ_Paletky),ADR(RFID_Hlava_2.PAR.PrecitaneCisloPaletky_POLE),SIZEOF(RFID_Hlava_2.PAR.PrecitaneCisloPaletky_POLE));

	//Rozdelenie prečítanej správy na číslo paletky a model//
	IF RFID_Hlava_2.STAV.PritomnostCipu THEN
		brsmemset(ADR(VstupnePoleUSINT),0,SIZEOF(VstupnePoleUSINT)); //Vymazanie vstupneho pola
		brsmemset(ADR(VystupnePoleStringov),0,SIZEOF(VystupnePoleStringov)); //Vymazanie výstupneho pola znakov
		PocetZnakovUDINT := brsstrlen(ADR(RFID_Hlava_2.PAR.Precitane_Cislo_Typ_Paletky)); //Zistenie počtu znakov vstupnej spravy
		PocetZnakovUSINT:= UDINT_TO_USINT(PocetZnakovUDINT);
		brsmemcpy(ADR(VstupnePoleUSINT),ADR(RFID_Hlava_2.PAR.Precitane_Cislo_Typ_Paletky),SIZEOF(RFID_Hlava_2.PAR.Precitane_Cislo_Typ_Paletky)); //Vyplnenie polia znakmy vstupnej správy
		h:= 1;
		FOR g:= 1 TO PocetZnakovUSINT BY 1 DO
			IF VstupnePoleUSINT[g] <> 59 THEN //59 je oddelovací znak bodkočiarka
				AktualNacitanyZnak:= VstupnePoleUSINT[g];
				brsstrcat(ADR(VystupnePoleStringov[h]),ADR(AktualNacitanyZnak));
			ELSE
				h:= h + 1;
			END_IF
		END_FOR
		RFID_Hlava_2.PAR.PrecitaneCisloPaletky:= VystupnePoleStringov[1];
		RFID_Hlava_2.PAR.PrecitanyTypPaletky:= VystupnePoleStringov[2];
	ELSE
		RFID_Hlava_2.PAR.PrecitaneCisloPaletky:= '';
		RFID_Hlava_2.PAR.PrecitanyTypPaletky:= '';
	END_IF

	CASE SC_Hlava_2.Step OF

		0:
			SC_Hlava_2.StepName:= '0 - Nulovanie';
			RFID_Hlava_2.CMD.CitajDATA:= FALSE;
			RFID_Hlava_2.CMD.ZapisDATA:= FALSE;
			RFID_Hlava_2.CMD.CitaciuHlavu_VYPNI:= FALSE;
			RFID_Hlava_2.OUT.Bit_AV:= FALSE;
			RFID_Hlava_2.OUT.Bit_GR:= FALSE;
			RFID_Hlava_2.OUT.Bit_TI:= FALSE;
			RFID_Hlava_2.OUT.Bit_KA:= FALSE;

			IF RFID_Hlava_2.STAV.PritomnostCipu THEN
				SC_Hlava_2.ResetStep:= TRUE;
				SC_Hlava_2.Step:= 1;
			END_IF

		1:
			SC_Hlava_2.StepName:= '1 - Rozhodnutie o cinnosti';
			IF NOT RFID_Hlava_2.STAV.PritomnostCipu THEN
				SC_Hlava_2.Step:= 0;
			ELSIF RFID_Hlava_2.CMD.CitajDATA THEN
				RFID_Hlava_2.STAV.CitanieDat_OK:= FALSE;
				RFID_Hlava_2.STAV.CitanieDat_ERROR:= FALSE;
				SC_Hlava_2.Step:= 10;
			ELSIF RFID_Hlava_2.CMD.ZapisDATA THEN
				RFID_Hlava_2.STAV.ZapisDat_OK:= FALSE;
				RFID_Hlava_2.STAV.ZapisDat_ERROR:= FALSE;
				SC_Hlava_2.Step:= 20;
			ELSIF RFID_Hlava_2.CMD.CitaciuHlavu_VYPNI THEN
				SC_Hlava_2.Step:= 30;
			END_IF

		10:
			SC_Hlava_2.StepName:= '10 - Citanie dat';
			SC_Hlava_2.IdleTime.PT:= T#3s;
			SC_Hlava_2.AlarmTime.PT:= T#6s;

			RFID_Hlava_2.IN.Old_Bit_TO:= RFID_Hlava_2.IN.Bit_TO;
			RFID_Hlava_2.OUT.BYTE_OUT[1]:= 1; //Kommand - 1 - čítanie, 2 - zápis
			RFID_Hlava_2.OUT.BYTE_OUT[2]:= 0; //Štartovacia adresa čítania (LSB) - na 2 byte začína zapisovať načítané znaky
			RFID_Hlava_2.OUT.BYTE_OUT[3]:= 0; //Štartovacia adresa čítania (HSB)
			RFID_Hlava_2.OUT.BYTE_OUT[4]:= 10; //Počet bajtov čítania (LSB) - 10 znakov
			RFID_Hlava_2.OUT.BYTE_OUT[5]:= 0; //Počet bajtov čítania (HSB)
			RFID_Hlava_2.OUT.Bit_AV:= TRUE;

			SC_Hlava_2.ResetStep:= TRUE;
			SC_Hlava_2.Step:= 11;

		11:
			SC_Hlava_2.StepName:= '11 - Citanie dat';
			SC_Hlava_2.IdleTime.PT:= T#3s;
			SC_Hlava_2.AlarmTime.PT:= T#2s;

			IF RFID_Hlava_2.IN.Bit_AA AND RFID_Hlava_2.IN.Bit_AE AND (RFID_Hlava_2.IN.Old_Bit_TO <> RFID_Hlava_2.IN.Bit_TO) THEN
				RFID_Hlava_2.STAV.CitanieDat_OK:= TRUE;
				SC_Hlava_2.ResetStep:= TRUE;
				SC_Hlava_2.Step:= 12;
			ELSIF RFID_Hlava_2.IN.Bit_AF THEN
				RFID_Hlava_2.STAV.CitanieDat_ERROR:= TRUE;
				SC_Hlava_2.ResetStep:= TRUE;
				SC_Hlava_2.Step:= 12;
			END_IF

		12:
			SC_Hlava_2.StepName:= '12 - Citanie dat';
			SC_Hlava_2.IdleTime.PT:= T#3s;
			SC_Hlava_2.AlarmTime.PT:= T#6s;

			RFID_Hlava_2.OUT.Bit_AV:= FALSE;

			IF NOT RFID_Hlava_2.IN.Bit_AA AND NOT RFID_Hlava_2.IN.Bit_AE AND NOT RFID_Hlava_2.IN.Bit_AF THEN
				SC_Hlava_2.ResetStep:= TRUE;
				SC_Hlava_2.Step:= 0;
			END_IF

		20:
			SC_Hlava_2.StepName:= '20 - Zápis dat';
			SC_Hlava_2.IdleTime.PT:= T#3s;
			SC_Hlava_2.AlarmTime.PT:= T#6s;

			RFID_Hlava_2.IN.Old_Bit_TO:= RFID_Hlava_2.IN.Bit_TO;
			RFID_Hlava_2.OUT.BYTE_OUT[1]:= 2; //Kommand - 1 - čítanie, 2 - zápis
			RFID_Hlava_2.OUT.BYTE_OUT[2]:= 0; //Štartovacia adresa zápisu (LSB) - na 2 byte začína zapisovať znaky
			RFID_Hlava_2.OUT.BYTE_OUT[3]:= 0; //Štartovacia adresa zápisu (HSB)
			RFID_Hlava_2.OUT.BYTE_OUT[4]:= 10; //Počet bajtov zápisu (LSB) - 10 znakov
			RFID_Hlava_2.OUT.BYTE_OUT[5]:= 0; //Počet bajtov zápisu (HSB)
			RFID_Hlava_2.OUT.Bit_AV:= TRUE;

			SC_Hlava_2.ResetStep:= TRUE;
			SC_Hlava_2.Step:= 21;

		21:
			SC_Hlava_2.StepName:= '21 - Zápis dat';
			SC_Hlava_2.IdleTime.PT:= T#3s;
			SC_Hlava_2.AlarmTime.PT:= T#2s;

			IF RFID_Hlava_2.IN.Bit_AA AND (RFID_Hlava_2.IN.Old_Bit_TO <> RFID_Hlava_2.IN.Bit_TO) THEN
				SC_Hlava_2.ResetStep:= TRUE;
				SC_Hlava_2.Step:= 22;
			END_IF

		22:
			SC_Hlava_2.StepName:= '21 - Zápis dat';
			SC_Hlava_2.IdleTime.PT:= T#3s;
			SC_Hlava_2.AlarmTime.PT:= T#6s;

			brsstrcpy(ADR(RFID_Hlava_2.PAR.ZadaneCisloPaletky_POLE),ADR(RFID_Hlava_2.PAR.Zadane_Cislo_Typ_Paletky));
			RFID_Hlava_2.OUT.BYTE_OUT[1]:= RFID_Hlava_2.PAR.ZadaneCisloPaletky_POLE[0];
			RFID_Hlava_2.OUT.BYTE_OUT[2]:= RFID_Hlava_2.PAR.ZadaneCisloPaletky_POLE[1];
			RFID_Hlava_2.OUT.BYTE_OUT[3]:= RFID_Hlava_2.PAR.ZadaneCisloPaletky_POLE[2];
			RFID_Hlava_2.OUT.BYTE_OUT[4]:= RFID_Hlava_2.PAR.ZadaneCisloPaletky_POLE[3];
			RFID_Hlava_2.OUT.BYTE_OUT[5]:= RFID_Hlava_2.PAR.ZadaneCisloPaletky_POLE[4];
			RFID_Hlava_2.OUT.BYTE_OUT[6]:= RFID_Hlava_2.PAR.ZadaneCisloPaletky_POLE[5];
			RFID_Hlava_2.OUT.BYTE_OUT[7]:= RFID_Hlava_2.PAR.ZadaneCisloPaletky_POLE[6];
			RFID_Hlava_2.OUT.BYTE_OUT[8]:= RFID_Hlava_2.PAR.ZadaneCisloPaletky_POLE[7];
			RFID_Hlava_2.OUT.BYTE_OUT[9]:= RFID_Hlava_2.PAR.ZadaneCisloPaletky_POLE[8];
			RFID_Hlava_2.OUT.BYTE_OUT[10]:= RFID_Hlava_2.PAR.ZadaneCisloPaletky_POLE[9];

			IF RFID_Hlava_2.OUT.Bit_TI THEN
				RFID_Hlava_2.OUT.Bit_TI:= FALSE;
				SC_Hlava_2.ResetStep:= TRUE;
				SC_Hlava_2.Step:= 23;
			ELSE
				RFID_Hlava_2.OUT.Bit_TI:= TRUE;
				SC_Hlava_2.ResetStep:= TRUE;
				SC_Hlava_2.Step:= 23;
			END_IF

		23:
			SC_Hlava_2.StepName:= '23 - Zápis dat';
			SC_Hlava_2.IdleTime.PT:= T#3s;
			SC_Hlava_2.AlarmTime.PT:= T#2s;

			IF RFID_Hlava_2.IN.Bit_AE THEN
				RFID_Hlava_2.STAV.ZapisDat_OK:= TRUE;
				SC_Hlava_2.ResetStep:= TRUE;
				SC_Hlava_2.Step:= 24;
			ELSIF RFID_Hlava_2.IN.Bit_AF THEN
				RFID_Hlava_2.STAV.ZapisDat_ERROR:= TRUE;
				SC_Hlava_2.ResetStep:= TRUE;
				SC_Hlava_2.Step:= 24;
			END_IF

		24:
			SC_Hlava_2.StepName:= '22 - Zápis dat';
			SC_Hlava_2.IdleTime.PT:= T#3s;
			SC_Hlava_2.AlarmTime.PT:= T#6s;

			RFID_Hlava_2.OUT.Bit_AV:= FALSE;

			IF NOT RFID_Hlava_2.IN.Bit_AA AND NOT RFID_Hlava_2.IN.Bit_AE AND NOT RFID_Hlava_2.IN.Bit_AF THEN
				SC_Hlava_2.ResetStep:= TRUE;
				SC_Hlava_2.Step:= 0;
			END_IF

		30:
			SC_Hlava_2.StepName:= '30 - Vypnutie citacej hlavy';
			SC_Hlava_2.IdleTime.PT:= T#3s;
			SC_Hlava_2.AlarmTime.PT:= T#2s;

			RFID_Hlava_2.OUT.Bit_KA:= TRUE;

			IF NOT RFID_Hlava_2.CMD.CitaciuHlavu_VYPNI THEN
				SC_Hlava_2.ResetStep:= TRUE;
				SC_Hlava_2.Step:= 0;
			END_IF

	END_CASE

END_ACTION
```

#### OvlTlaciarne.st
```iecst
ACTION OvlTlaciarne:

	//SATO parametre komunikácie//
	//IP: 192.168.1.6
	//255.255.255.0
	//Port č.:9100

	PrvyRiadok:= 'A5E30093844AACO';
	DruhyRiadok:= 'A5E30093844AACO@210722B0106';
	TretiRiadok:= '07/2021';
	DataMetrix:= DruhyRiadok;

		//**************************************Textové polia etikety**************************************//

	//Správa pre tlačiareň SATO HR224R//
	Tlaciaren.Data.Sprava_pre_Tlaciaren:= 'A';//Začiatok správy
	strcat(ADR(Tlaciaren.Data.Sprava_pre_Tlaciaren),ADR('%0')); //rotácia textu 0 - 0°, 1 - 90°, 2 - 180°, 3 - 270°
	strcat(ADR(Tlaciaren.Data.Sprava_pre_Tlaciaren),ADR('A103600840')); //rozmer etikety výška 0360/24 = 15mm, šírka 0840/24 = 35mm
	strcat(ADR(Tlaciaren.Data.Sprava_pre_Tlaciaren),ADR('V0012')); //posunutie textu vertikálne
	strcat(ADR(Tlaciaren.Data.Sprava_pre_Tlaciaren),ADR('H0055')); //posunutie textu horizontálne
	strcat(ADR(Tlaciaren.Data.Sprava_pre_Tlaciaren),ADR('P2')); //velkost medzery medzi pismenami
	strcat(ADR(Tlaciaren.Data.Sprava_pre_Tlaciaren),ADR('L0710')); //násobok velkosti písma
	strcat(ADR(Tlaciaren.Data.Sprava_pre_Tlaciaren),ADR('U'));
	strcat(ADR(Tlaciaren.Data.Sprava_pre_Tlaciaren),ADR(PrvyRiadok));
	strcat(ADR(Tlaciaren.Data.Sprava_pre_Tlaciaren),ADR('V0098')); //posunutie textu vertikálne
	strcat(ADR(Tlaciaren.Data.Sprava_pre_Tlaciaren),ADR('H0055')); //posunutie textu horizontálne
	strcat(ADR(Tlaciaren.Data.Sprava_pre_Tlaciaren),ADR('P2')); //velkost medzery medzi pismenami
	strcat(ADR(Tlaciaren.Data.Sprava_pre_Tlaciaren),ADR('L0406')); //násobok velkosti písma
	strcat(ADR(Tlaciaren.Data.Sprava_pre_Tlaciaren),ADR('U'));
	strcat(ADR(Tlaciaren.Data.Sprava_pre_Tlaciaren),ADR(DruhyRiadok));
	strcat(ADR(Tlaciaren.Data.Sprava_pre_Tlaciaren),ADR('V0216')); //posunutie textu vertikálne
	strcat(ADR(Tlaciaren.Data.Sprava_pre_Tlaciaren),ADR('H0312')); //posunutie textu horizontálne
	strcat(ADR(Tlaciaren.Data.Sprava_pre_Tlaciaren),ADR('P2')); //velkost medzery medzi pismenami
	strcat(ADR(Tlaciaren.Data.Sprava_pre_Tlaciaren),ADR('L0609')); //násobok velkosti písma
	strcat(ADR(Tlaciaren.Data.Sprava_pre_Tlaciaren),ADR('U'));
	strcat(ADR(Tlaciaren.Data.Sprava_pre_Tlaciaren),ADR(TretiRiadok));
	strcat(ADR(Tlaciaren.Data.Sprava_pre_Tlaciaren),ADR('V0168')); //posunutie textu vertikálne
	strcat(ADR(Tlaciaren.Data.Sprava_pre_Tlaciaren),ADR('H0055')); //posunutie textu horizontálne
	strcat(ADR(Tlaciaren.Data.Sprava_pre_Tlaciaren),ADR('BX01201010000000001')); //Definícia Datametrixu
	strcat(ADR(Tlaciaren.Data.Sprava_pre_Tlaciaren),ADR('DC'));
	strcat(ADR(Tlaciaren.Data.Sprava_pre_Tlaciaren),ADR(DataMetrix));
	strcat(ADR(Tlaciaren.Data.Sprava_pre_Tlaciaren),ADR('Q1')); //Počet výtlačkov etikety
	strcat(ADR(Tlaciaren.Data.Sprava_pre_Tlaciaren),ADR('Z'));//Koniec správy

	//Hodnotu vydelíme 24 aby sme dostali vzdialenost v mm//

END_ACTION
```

### Program Logical/Program/Robot (IEC)

#### Main.st - Init, cyclic, exit code
```iecst
PROGRAM _INIT
	(* Insert code here *)

END_PROGRAM

PROGRAM _CYCLIC

	//Volanie podprogramov//
	KOM_Robot;
	KOM_Kamera;

	//Volanie funkcie SequenceControl//
	SequenceControl(SC:= SC_Robot);

	//Reset sekcie //
	IF Robot.Reset THEN
		SC_Robot.Step:= 0;
		Robot.Reset:= FALSE;
	ELSIF NOT Safety.STAV.ZonaCS_AKTIVNA  THEN
		SC_Robot.Step:= 0;
	ELSIF Robot.Automat AND (NOT Safety.STAV.BarieraDopravnikaNG_AKTIVNA AND NOT Safety.STAV.MutingRobota_AKTIVNY) THEN
		Alarmy[72]:= TRUE;
		SC_Robot.Step:= 0;
		SC_StoperEtiketovania.Step:= 0;
		PoruchaBunky:= TRUE;
	ELSIF Robot.Automat AND NOT Safety.STAV.ServisneDvereTlaciarne_AKTIVNE THEN
		Alarmy[71]:= TRUE;
		SC_Robot.Step:= 0;
		SC_StoperEtiketovania.Step:= 0;
		PoruchaBunky:= TRUE;
	END_IF

	CASE SC_Robot.Step OF

		0:
			SC_Robot.StepName:='0 - Nulovanie';
			Robot.Automat:= FALSE;
			Robot.KoniecCyklu:= FALSE;
			Robot.Manual:= FALSE;
			Robot.STAV.PoINIT:= FALSE;
			Robot.KOM_OUT.OdparkujRobota:= FALSE;
			Robot.KOM_OUT.PP_na_Main:= FALSE;
			Robot.KOM_OUT.Reset_CS:= FALSE;
			Robot.KOM_OUT.StartProgramu:= FALSE;
			Robot.KOM_OUT.StartProgramuMain:= FALSE;
			Robot.KOM_OUT.VypniMotory:= FALSE;
			Robot.KOM_OUT.ZapniMotory:= FALSE;
			Robot.Odparkovanie:= FALSE;
			Robot.KOM_OUT.PresunDoPozicieOdobratiaEtikety:= FALSE;
			Robot.KOM_OUT.PresunDoMutingPozicie:= FALSE;
			Robot.KOM_OUT.PresunDoPoziceKontrolyEtikety:= FALSE;
			Robot.KOM_OUT.PresunDoPoziceKontrEtiketyPriamo:= FALSE;
			Robot.KOM_OUT.PresunDoPozicieKontrolyIntStitku:= FALSE;
			Robot.KOM_OUT.NalepEtiketu:= FALSE;
			Robot.KOM_OUT.CitanieStitkuUkoncene:= FALSE;
			Robot.RR_PresunPoziciaCitaniaDMkodu:= FALSE;
			Robot.RR_PresunPoziciaCitaniaQRkodu:= FALSE;
			Robot.RR_PresunPoziciaNalepeniaEtikety:= FALSE;
			Robot.RR_PresunPoziciaOdobratiaEtikety:= FALSE;

			IF Robot.KOM_IN.Stav_RezimAUTOMAT AND Robot.KOM_IN.Stav_ProgramRUN THEN
				Robot.KOM_OUT.StopProgramu:= TRUE;
			ELSE
				Robot.KOM_OUT.StopProgramu:= FALSE;
			END_IF
			IF Safety.STAV.ZonaCS_AKTIVNA AND Safety.STAV.ZonaBunky_AKTIVNA AND Linka.IN.TlakVzduchu_OK_S2 AND NOT NastalaPorucha AND NOT Robot.KOM_IN.Stav_ProgramRUN AND Linka.STAV.Hardware_OK THEN
				Robot.KOM_OUT.StopProgramu:= FALSE;
				SC_Robot.ResetStep:= TRUE;
				SC_Robot.Step:= 1;
			END_IF

		1:
			SC_Robot.StepName:='1 - Cakam na spustenie vyroby';
			Robot.KoniecCyklu:= FALSE;
			IF Robot.Automat THEN
				SC_Robot.Step:= 2;
			ELSIF Robot.Odparkovanie THEN
				SC_Robot.Step:= 2;
			ELSIF Robot.RR_PresunPoziciaCitaniaQRkodu THEN
				Robot.Manual:= TRUE;
				SC_Robot.Step:= 2;
			ELSIF Robot.RR_PresunPoziciaCitaniaDMkodu THEN
				Robot.Manual:= TRUE;
				SC_Robot.Step:= 2;
			ELSIF Robot.RR_PresunPoziciaOdobratiaEtikety THEN
				Robot.Manual:= TRUE;
				SC_Robot.Step:= 2;
			END_IF

			//********************************************************Inicializácia****************************************************************************//

		2:
			SC_Robot.StepName:='2 - Inicializacia - cakam na spustenie inicializacie';
			SC_Robot.IdleTime.PT:= T#500ms;
			SC_Robot.AlarmTime.PT:= T#5s;

			SC_Robot.IdleTime.IN:= TRUE;

			IF SC_Robot.IdleTime.Q THEN
				SC_Robot.ResetStep:= TRUE;
				SC_Robot.Step:= 3;
			END_IF

		3:
			SC_Robot.StepName:='2 - Inicializacia - kontrolujem central stop robota';
			SC_Robot.IdleTime.PT:= T#500ms;
			SC_Robot.AlarmTime.PT:= T#5s;

			IF Robot.KOM_IN.Stav_RobotCS THEN
				Robot.KOM_OUT.Reset_CS:= TRUE;
			END_IF

			IF NOT Robot.KOM_IN.Stav_RobotCS THEN
				Robot.KOM_OUT.Reset_CS:= FALSE;
				SC_Robot.ResetStep:= TRUE;
				SC_Robot.Step:= 4;
			END_IF

		4:
			SC_Robot.StepName:='4 - Inicializacia - zapinam motory robota';
			SC_Robot.IdleTime.PT:= T#500ms;
			SC_Robot.AlarmTime.PT:= T#5s;

			IF NOT Robot.KOM_IN.Stav_MotoryON THEN
				Robot.KOM_OUT.ZapniMotory:= TRUE;
			END_IF

			IF Robot.KOM_IN.Stav_MotoryON THEN
				Robot.KOM_OUT.ZapniMotory:= FALSE;
				SC_Robot.ResetStep:= TRUE;
				SC_Robot.Step:= 6;
			END_IF

		6:
			SC_Robot.StepName:='6 - Inicializacia - spustam program robota od zaciatku';
			SC_Robot.IdleTime.PT:= T#500ms;
			SC_Robot.AlarmTime.PT:= T#5s;

			IF NOT SC_Robot.Switch1 THEN
				Robot.KOM_OUT.StartProgramuMain:= TRUE;
				SC_Robot.Switch1:= TRUE;
			END_IF

			IF Robot.KOM_IN.Stav_ProgramRUN AND Robot.KOM_IN.Stav_VystupyZresetovane THEN
				Robot.KOM_OUT.StartProgramuMain:= FALSE;
				IF Robot.RR_PresunPoziciaCitaniaQRkodu THEN
					SC_Robot.ResetStep:= TRUE;
					SC_Robot.Step:= 700;
				ELSIF Robot.RR_PresunPoziciaCitaniaDMkodu THEN
					SC_Robot.ResetStep:= TRUE;
					SC_Robot.Step:= 720;
				ELSIF Robot.RR_PresunPoziciaOdobratiaEtikety THEN
					SC_Robot.ResetStep:= TRUE;
					SC_Robot.Step:= 740;
				ELSIF Robot.Odparkovanie AND Safety.STAV.MutingRobota_AKTIVNY THEN
					SC_Robot.ResetStep:= TRUE;
					SC_Robot.Step:= 0;
				ELSIF NOT Robot.Odparkovanie THEN
					Robot.STAV.PoINIT:= TRUE;
					SC_Robot.ResetStep:= TRUE;
					SC_Robot.Step:= 100;
				END_IF
			END_IF

			//********************************************************Automatický režim****************************************************************************//

		100:
			SC_Robot.StepName:='100 - Automaticky Rezim - cakam na ukoncenie programu robota';
			SC_Robot.IdleTime.PT:= T#200ms;
			SC_Robot.AlarmTime.PT:= T#5s;

			IF NOT Robot.KOM_IN.Stav_ProgramRUN THEN
				Alarmy[73]:= TRUE;
				PoruchaBunky:= TRUE;
				SC_Robot.ResetStep:= TRUE;
				SC_Robot.Step:= 0;
			ELSIF Robot.KoniecCyklu AND NOT StoperEtiketovania.Automat AND NOT StoperDopravNG.Automat THEN
				SC_Robot.ResetStep:= TRUE;
				SC_Robot.Step:= 0;
			END_IF

			//*******************************************************Manuálny režim*******************************************************************************//

		700:
			SC_Robot.StepName:='700 - Manualny Rezim - citania QR kodu internej etikety,precitanie typu paletky,zvolenie cisla programu pre robot a cisla programu kamery';
			SC_Robot.IdleTime.PT:= T#200ms;
			SC_Robot.AlarmTime.PT:= T#5s;

			SC_Robot.IdleTime.IN:= RFID_Hlava_2.STAV.PritomnostCipu;

			IF NOT RFID_Hlava_2.STAV.PritomnostCipu THEN
				SC_Robot.ResetStep:= TRUE;
				SC_Robot.Step:= 0;
			ELSIF SC_Robot.IdleTime.Q THEN
				IF RFID_Hlava_2.PAR.PrecitaneCisloPaletky <> '' AND Linka.PAR.Zvoleny_MODEL <> '' THEN
					IF RFID_Hlava_2.PAR.PrecitanyTypPaletky = 'BF1' AND Linka.PAR.Zvoleny_MODEL = 'EZTKB24380HA' THEN
						Robot.KOM_OUT.CisloProduktu:= 1;
						IF Kamera.STAV.AktualneCisloProgramu <> 1 THEN
							Kamera.PAR.ZadaneCisloProgramu:= 1;
						END_IF
					ELSIF RFID_Hlava_2.PAR.PrecitanyTypPaletky = 'BV1' THEN
						Robot.KOM_OUT.CisloProduktu:= 2;
						IF Kamera.STAV.AktualneCisloProgramu <> 3 THEN
							Kamera.PAR.ZadaneCisloProgramu:= 3;
						END_IF
					ELSIF RFID_Hlava_2.PAR.PrecitanyTypPaletky = 'BW1' THEN
						Robot.KOM_OUT.CisloProduktu:= 3;
						IF Kamera.STAV.AktualneCisloProgramu <> 5 THEN
							Kamera.PAR.ZadaneCisloProgramu:= 5;
						END_IF
					ELSIF RFID_Hlava_2.PAR.PrecitanyTypPaletky = 'CN1' THEN
						Robot.KOM_OUT.CisloProduktu:= 4;
						IF Kamera.STAV.AktualneCisloProgramu <> 7 THEN
							Kamera.PAR.ZadaneCisloProgramu:= 7;
						END_IF
					ELSIF RFID_Hlava_2.PAR.PrecitanyTypPaletky = 'CP1' THEN
						Robot.KOM_OUT.CisloProduktu:= 5;
						IF Kamera.STAV.AktualneCisloProgramu <> 9 THEN
							Kamera.PAR.ZadaneCisloProgramu:= 9;
						END_IF
					ELSIF RFID_Hlava_2.PAR.PrecitanyTypPaletky = 'BE1' THEN
						Robot.KOM_OUT.CisloProduktu:= 6;
						Kamera.PAR.ZadaneCisloProgramu:= 11;
					ELSIF RFID_Hlava_2.PAR.PrecitanyTypPaletky = 'BD1' THEN
						Robot.KOM_OUT.CisloProduktu:= 7;
						IF Kamera.STAV.AktualneCisloProgramu <> 13 THEN
							Kamera.PAR.ZadaneCisloProgramu:= 13;
						END_IF
					ELSIF RFID_Hlava_2.PAR.PrecitanyTypPaletky = 'BF1' AND Linka.PAR.Zvoleny_MODEL = 'EZTYB21670HA' THEN
						Robot.KOM_OUT.CisloProduktu:= 8;
						IF Kamera.STAV.AktualneCisloProgramu <> 15 THEN
							Kamera.PAR.ZadaneCisloProgramu:= 15;
						END_IF
					ELSE
						SC_Robot.ResetStep:= TRUE;
						SC_Robot.Step:= 0;
					END_IF
					SC_Robot.ResetStep:= TRUE;
					SC_Robot.Step:= 701;
				ELSE
					SC_Robot.ResetStep:= TRUE;
					SC_Robot.Step:= 0;
				END_IF
			END_IF

		701:
			SC_Robot.StepName:='701 - Manualny Rezim - zacentrovanie paletky';
			SC_Robot.IdleTime.PT:= T#200ms;
			SC_Robot.AlarmTime.PT:= T#5s;

			IF NOT SC_Robot.Switch1 THEN
				StoperEtiketovania.RR_ZacentrujPaletku:= TRUE;
				SC_Robot.Switch1:= TRUE;
			END_IF

			IF StoperEtiketovania.IN.Centrovanie_HornaPoloha_IS18 THEN
				SC_Robot.ResetStep:= TRUE;
				SC_Robot.Step:= 702;
			END_IF

		702:
			SC_Robot.StepName:='702 - Manualny Rezim - citania QR kodu internej etikety,presun robota do pozicie citania internej etikety';
			SC_Robot.IdleTime.PT:= T#200ms;
			SC_Robot.AlarmTime.PT:= T#5s;

			IF NOT SC_Robot.Switch1 THEN
				Robot.KOM_OUT.PresunDoPozicieKontrolyIntStitku:= TRUE;
				SC_Robot.Switch1:= TRUE;
			END_IF

			IF Robot.KOM_IN.Stav_RobotCinnostUkoncena THEN
				Robot.KOM_OUT.PresunDoPozicieKontrolyIntStitku:= FALSE;
				SC_Robot.ResetStep:= TRUE;
				SC_Robot.Step:= 705;
			END_IF

		705:
			SC_Robot.StepName:='705 - Manualny Rezim - citania QR kodu internej etikety,cakam na zrusenie signalu cinnost robota ukoncena';
			SC_Robot.IdleTime.PT:= T#200ms;
			SC_Robot.AlarmTime.PT:= T#5s;

			IF NOT Robot.KOM_IN.Stav_RobotCinnostUkoncena THEN
				SC_Robot.ResetStep:= TRUE;
				SC_Robot.Step:= 708;
			END_IF

		708:
			SC_Robot.StepName:='708 - Manualny Rezim - citania QR kodu internej etikety,cakam na ukoncenie citania internej etikety';
			SC_Robot.IdleTime.PT:= T#200ms;
			SC_Robot.AlarmTime.PT:= T#5s;

			IF NOT SC_Robot.Switch1 AND NOT Robot.RR_PresunPoziciaCitaniaQRkodu THEN
				Robot.KOM_OUT.CitanieStitkuUkoncene:= TRUE;
				SC_Robot.Switch1:= TRUE;
			END_IF

			IF Robot.KOM_IN.Stav_RobotCinnostUkoncena THEN
				Robot.KOM_OUT.CitanieStitkuUkoncene:= FALSE;
				SC_Robot.ResetStep:= TRUE;
				SC_Robot.Step:= 710;
			END_IF

		710:
			SC_Robot.StepName:='710 - Manualny Rezim - citania QR kodu internej etikety,cakam na zrusenie signalu cinnost robota ukoncena';
			SC_Robot.IdleTime.PT:= T#200ms;
			SC_Robot.AlarmTime.PT:= T#5s;

			IF NOT Robot.KOM_IN.Stav_RobotCinnostUkoncena THEN
				SC_Robot.ResetStep:= TRUE;
				SC_Robot.Step:= 713;
			END_IF

		713:
			SC_Robot.StepName:='713 - Manualny Rezim - citania QR kodu internej etikety,presun robota do muting pozicie';
			SC_Robot.IdleTime.PT:= T#200ms;
			SC_Robot.AlarmTime.PT:= T#5s;

			IF NOT SC_Robot.Switch1 THEN
				Robot.KOM_OUT.PresunDoMutingPozicie:= TRUE;
				SC_Robot.Switch1:= TRUE;
			END_IF

			IF Robot.KOM_IN.Stav_RobotCinnostUkoncena AND Safety.STAV.MutingRobota_AKTIVNY THEN
				Robot.KOM_OUT.PresunDoMutingPozicie:= FALSE;
				SC_Robot.ResetStep:= TRUE;
				SC_Robot.Step:= 714;
			END_IF

		714:
			SC_Robot.StepName:='714 - Manualny Rezim - odcentrovanie paletky';
			SC_Robot.IdleTime.PT:= T#200ms;
			SC_Robot.AlarmTime.PT:= T#5s;

			IF NOT SC_Robot.Switch1 AND NOT Robot.KOM_IN.Stav_RobotCinnostUkoncena THEN
				StoperEtiketovania.RR_OdcentrujPaletku:= TRUE;
				SC_Robot.Switch1:= TRUE;
			END_IF

			IF StoperEtiketovania.IN.Centrovanie_SpodnaPoloha_IS17 THEN
				SC_Robot.ResetStep:= TRUE;
				SC_Robot.Step:= 0;
			END_IF

		720:
			SC_Robot.StepName:='720 - Manualny Rezim - citania DM kodu zakaznickej etikety,precitanie typu paletky,zvolenie cisla programu pre robot a cisla programu kamery';
			SC_Robot.IdleTime.PT:= T#200ms;
			SC_Robot.AlarmTime.PT:= T#5s;

			SC_Robot.IdleTime.IN:= RFID_Hlava_2.STAV.PritomnostCipu;

			IF NOT RFID_Hlava_2.STAV.PritomnostCipu THEN
				SC_Robot.ResetStep:= TRUE;
				SC_Robot.Step:= 0;
			ELSIF SC_Robot.IdleTime.Q THEN
				IF RFID_Hlava_2.PAR.PrecitaneCisloPaletky <> '' AND Linka.PAR.Zvoleny_MODEL <> '' THEN
					IF RFID_Hlava_2.PAR.PrecitanyTypPaletky = 'BF1' AND Linka.PAR.Zvoleny_MODEL = 'EZTKB24380HA' THEN
						Robot.KOM_OUT.CisloProduktu:= 1;
						IF Kamera.STAV.AktualneCisloProgramu <> 2 THEN
							Kamera.PAR.ZadaneCisloProgramu:= 2;
						END_IF
					ELSIF RFID_Hlava_2.PAR.PrecitanyTypPaletky = 'BV1' THEN
						Robot.KOM_OUT.CisloProduktu:= 2;
						IF Kamera.STAV.AktualneCisloProgramu <> 4 THEN
							Kamera.PAR.ZadaneCisloProgramu:= 4;
						END_IF
					ELSIF RFID_Hlava_2.PAR.PrecitanyTypPaletky = 'BW1' THEN
						Robot.KOM_OUT.CisloProduktu:= 3;
						IF Kamera.STAV.AktualneCisloProgramu <> 6 THEN
							Kamera.PAR.ZadaneCisloProgramu:= 6;
						END_IF
					ELSIF RFID_Hlava_2.PAR.PrecitanyTypPaletky = 'CN1' THEN
						Robot.KOM_OUT.CisloProduktu:= 4;
						IF Kamera.STAV.AktualneCisloProgramu <> 8 THEN
							Kamera.PAR.ZadaneCisloProgramu:= 8;
						END_IF
					ELSIF RFID_Hlava_2.PAR.PrecitanyTypPaletky = 'CP1' THEN
						Robot.KOM_OUT.CisloProduktu:= 5;
						IF Kamera.STAV.AktualneCisloProgramu <> 10 THEN
							Kamera.PAR.ZadaneCisloProgramu:= 10;
						END_IF
					ELSIF RFID_Hlava_2.PAR.PrecitanyTypPaletky = 'BE1' THEN
						Robot.KOM_OUT.CisloProduktu:= 6;
						IF Kamera.STAV.AktualneCisloProgramu <> 12 THEN
							Kamera.PAR.ZadaneCisloProgramu:= 12;
						END_IF
					ELSIF RFID_Hlava_2.PAR.PrecitanyTypPaletky = 'BD1' THEN
						Robot.KOM_OUT.CisloProduktu:= 7;
						IF Kamera.STAV.AktualneCisloProgramu <> 14 THEN
							Kamera.PAR.ZadaneCisloProgramu:= 14;
						END_IF
					ELSIF RFID_Hlava_2.PAR.PrecitanyTypPaletky = 'BF1' AND Linka.PAR.Zvoleny_MODEL = 'EZTYB21670HA' THEN
						Robot.KOM_OUT.CisloProduktu:= 8;
						IF Kamera.STAV.AktualneCisloProgramu <> 16 THEN
							Kamera.PAR.ZadaneCisloProgramu:= 16;
						END_IF
					ELSE
						SC_Robot.ResetStep:= TRUE;
						SC_Robot.Step:= 0;
					END_IF
					SC_Robot.ResetStep:= TRUE;
					SC_Robot.Step:= 721;
				ELSE
					SC_Robot.ResetStep:= TRUE;
					SC_Robot.Step:= 0;
				END_IF
			END_IF

		721:
			SC_Robot.StepName:='721 - Manualny Rezim - zacentrovanie paletky';
			SC_Robot.IdleTime.PT:= T#200ms;
			SC_Robot.AlarmTime.PT:= T#5s;

			IF NOT SC_Robot.Switch1 THEN
				StoperEtiketovania.RR_ZacentrujPaletku:= TRUE;
				SC_Robot.Switch1:= TRUE;
			END_IF

			IF StoperEtiketovania.IN.Centrovanie_HornaPoloha_IS18 THEN
				SC_Robot.ResetStep:= TRUE;
				SC_Robot.Step:= 722;
			END_IF

		722:
			SC_Robot.StepName:='722 - Manualny Rezim - citania DM kodu zakaznickej etikety,presun robota do pozicie citania zakaznickej etikety';
			SC_Robot.IdleTime.PT:= T#200ms;
			SC_Robot.AlarmTime.PT:= T#5s;

			IF NOT SC_Robot.Switch1 THEN
				Robot.KOM_OUT.PresunDoPoziceKontrEtiketyPriamo:= TRUE;
				SC_Robot.Switch1:= TRUE;
			END_IF

			IF Robot.KOM_IN.Stav_RobotCinnostUkoncena THEN
				Robot.KOM_OUT.PresunDoPoziceKontrEtiketyPriamo:= FALSE;
				SC_Robot.ResetStep:= TRUE;
				SC_Robot.Step:= 725;
			END_IF

		725:
			SC_Robot.StepName:='725 - Manualny Rezim - citania DM kodu zakaznickej etikety,cakam na zrusenie signalu cinnost robota ukoncena';
			SC_Robot.IdleTime.PT:= T#200ms;
			SC_Robot.AlarmTime.PT:= T#5s;

			IF NOT Robot.KOM_IN.Stav_RobotCinnostUkoncena THEN
				SC_Robot.ResetStep:= TRUE;
				SC_Robot.Step:= 728;
			END_IF

		728:
			SC_Robot.StepName:='728 - Manualny Rezim - citania DM kodu zakaznickej etikety,cakam na ukoncenie citania zakaznickej etikety';
			SC_Robot.IdleTime.PT:= T#200ms;
			SC_Robot.AlarmTime.PT:= T#5s;

			IF NOT SC_Robot.Switch1 AND NOT Robot.RR_PresunPoziciaCitaniaDMkodu THEN
				Robot.KOM_OUT.CitanieStitkuUkoncene:= TRUE;
				SC_Robot.Switch1:= TRUE;
			END_IF

			IF Robot.KOM_IN.Stav_RobotCinnostUkoncena THEN
				Robot.KOM_OUT.CitanieStitkuUkoncene:= FALSE;
				SC_Robot.ResetStep:= TRUE;
				SC_Robot.Step:= 730;
			END_IF

		730:
			SC_Robot.StepName:='730 - Manualny Rezim - citania DM kodu zakaznickej etikety,cakam na zrusenie signalu cinnost robota ukoncena';
			SC_Robot.IdleTime.PT:= T#200ms;
			SC_Robot.AlarmTime.PT:= T#5s;

			IF NOT Robot.KOM_IN.Stav_RobotCinnostUkoncena THEN
				SC_Robot.ResetStep:= TRUE;
				SC_Robot.Step:= 733;
			END_IF

		733:
			SC_Robot.StepName:='733 - Manualny Rezim - citania DM kodu zakaznickej etikety,presun robota do muting pozicie';
			SC_Robot.IdleTime.PT:= T#200ms;
			SC_Robot.AlarmTime.PT:= T#5s;

			IF NOT SC_Robot.Switch1 THEN
				Robot.KOM_OUT.PresunDoMutingPozicie:= TRUE;
				SC_Robot.Switch1:= TRUE;
			END_IF

			IF Robot.KOM_IN.Stav_RobotCinnostUkoncena AND Safety.STAV.MutingRobota_AKTIVNY THEN
				Robot.KOM_OUT.PresunDoMutingPozicie:= FALSE;
				SC_Robot.ResetStep:= TRUE;
				SC_Robot.Step:= 734;
			END_IF

		734:
			SC_Robot.StepName:='734 - Manualny Rezim - odcentrovanie paletky';
			SC_Robot.IdleTime.PT:= T#200ms;
			SC_Robot.AlarmTime.PT:= T#5s;

			IF NOT SC_Robot.Switch1 AND NOT Robot.KOM_IN.Stav_RobotCinnostUkoncena THEN
				StoperEtiketovania.RR_OdcentrujPaletku:= TRUE;
				SC_Robot.Switch1:= TRUE;
			END_IF

			IF StoperEtiketovania.IN.Centrovanie_SpodnaPoloha_IS17 THEN
				SC_Robot.ResetStep:= TRUE;
				SC_Robot.Step:= 0;
			END_IF

		740:
			SC_Robot.StepName:='740 - Manualny Rezim - presun robota do pozicie odobratia etikety z tlaciarne';
			SC_Robot.IdleTime.PT:= T#200ms;
			SC_Robot.AlarmTime.PT:= T#5s;

			IF NOT SC_Robot.Switch1 THEN
				Robot.KOM_OUT.PresunDoPozicieOdobratiaEtikety:= TRUE;
				SC_Robot.Switch1:= TRUE;
			END_IF

			IF Robot.KOM_IN.Stav_RobotCinnostUkoncena THEN
				Robot.KOM_OUT.PresunDoPozicieOdobratiaEtikety:= FALSE;
				SC_Robot.ResetStep:= TRUE;
				SC_Robot.Step:= 745;
			END_IF

		745:
			SC_Robot.StepName:='745 - Manualny Rezim - cakam na zrusenie signalu cinnost robota ukoncena';
			SC_Robot.IdleTime.PT:= T#200ms;
			SC_Robot.AlarmTime.PT:= T#5s;

			IF NOT Robot.KOM_IN.Stav_RobotCinnostUkoncena THEN
				SC_Robot.ResetStep:= TRUE;
				SC_Robot.Step:= 748;
			END_IF

		748:
			SC_Robot.StepName:='748 - Manualny Rezim - cakam na ukoncenie presunu odobratia etikety z tlaciarne';
			SC_Robot.IdleTime.PT:= T#200ms;
			SC_Robot.AlarmTime.PT:= T#5s;

			IF NOT SC_Robot.Switch1 AND NOT Robot.RR_PresunPoziciaOdobratiaEtikety THEN
				Robot.KOM_OUT.PresunDoMutingPozicie:= TRUE;
				SC_Robot.Switch1:= TRUE;
			END_IF

			IF Robot.KOM_IN.Stav_RobotCinnostUkoncena AND Safety.STAV.MutingRobota_AKTIVNY THEN
				Robot.KOM_OUT.PresunDoMutingPozicie:= FALSE;
				SC_Robot.ResetStep:= TRUE;
				SC_Robot.Step:= 750;
			END_IF

		750:
			SC_Robot.StepName:='750 - Manualny Rezim - cakam na zrusenie signalu cinnost robota ukoncena';
			SC_Robot.IdleTime.PT:= T#200ms;
			SC_Robot.AlarmTime.PT:= T#5s;

			IF NOT Robot.KOM_IN.Stav_RobotCinnostUkoncena THEN
				SC_Robot.ResetStep:= TRUE;
				SC_Robot.Step:= 0;
			END_IF

	END_CASE

END_PROGRAM

PROGRAM _EXIT
	(* Insert code here *)

END_PROGRAM
```

#### Variables.var - Local variables
```iecst
VAR
	PocetNacitZnakovQRkodu : UDINT := 0;
	PocetNacitZnakovDMkodu : UDINT := 0;
	CasPoPrepProgramuKamery : TON := (0);
	CasResetovaniaKamery : TON := (0);
END_VAR
```

#### KOM_Robot.st
```iecst
ACTION KOM_Robot:

	//Vstupy z Robota do PLC//
	Robot.KOM_IN.Stav_RezimAUTOMAT:= Robot.KOM_IN.Profinet_PLC_INPUTS[0].0;	                	//0
	Robot.KOM_IN.Stav_ProgramRUN:= Robot.KOM_IN.Profinet_PLC_INPUTS[0].1;                   	//1
	Robot.KOM_IN.Stav_MotoryOFF:= Robot.KOM_IN.Profinet_PLC_INPUTS[0].2;                    	//2
	Robot.KOM_IN.Stav_MotoryON:= Robot.KOM_IN.Profinet_PLC_INPUTS[0].3;                     	//3
	Robot.KOM_IN.Stav_RobotCS:= Robot.KOM_IN.Profinet_PLC_INPUTS[0].4;                      	//4
	Robot.KOM_IN.Profinet_PLC_INPUTS[0].5;                                                  	//5
	Robot.KOM_IN.Profinet_PLC_INPUTS[0].6;                                                  	//6
	Robot.KOM_IN.Profinet_PLC_INPUTS[0].7;														//7

	Robot.KOM_IN.Stav_RobotCinnostUkoncena:= Robot.KOM_IN.Profinet_PLC_INPUTS[1].0;				//8
	Robot.KOM_IN.Stav_RobotOdparkovany:= Robot.KOM_IN.Profinet_PLC_INPUTS[1].1;					//9
	Robot.KOM_IN.Stav_VystupyZresetovane:= Robot.KOM_IN.Profinet_PLC_INPUTS[1].2;				//10
	Prisavka_ON:= Robot.KOM_IN.Profinet_PLC_INPUTS[1].3;
	(*Robot.PrisavanieEtikety_ZAPNI:= Robot.KOM_IN.Profinet_PLC_INPUTS[1].3;*)						//11
	Robot.KOM_IN.Profinet_PLC_INPUTS[1].4;														//12
	Robot.KOM_IN.Profinet_PLC_INPUTS[1].5;														//13
	Robot.KOM_IN.Profinet_PLC_INPUTS[1].6;														//14
	Robot.KOM_IN.Profinet_PLC_INPUTS[1].7;  										 			//15

	Robot.KOM_IN.Profinet_PLC_INPUTS[2].0;														//16
	Robot.KOM_IN.Profinet_PLC_INPUTS[2].1;														//17
	Robot.KOM_IN.Profinet_PLC_INPUTS[2].2;														//18
	Robot.KOM_IN.Profinet_PLC_INPUTS[2].3;														//19
	Robot.KOM_IN.Profinet_PLC_INPUTS[2].4;														//20
	Robot.KOM_IN.Profinet_PLC_INPUTS[2].5;														//21
	Robot.KOM_IN.Profinet_PLC_INPUTS[2].6;														//22
	Robot.KOM_IN.Profinet_PLC_INPUTS[2].7;														//23

	Robot.KOM_IN.Profinet_PLC_INPUTS[3].0;														//24
	Robot.KOM_IN.Profinet_PLC_INPUTS[3].1;														//25
	Robot.KOM_IN.Profinet_PLC_INPUTS[3].2;														//26
	Robot.KOM_IN.Profinet_PLC_INPUTS[3].3;														//27
	Robot.KOM_IN.Profinet_PLC_INPUTS[3].4;														//28
	Robot.KOM_IN.Profinet_PLC_INPUTS[3].5;														//29
	Robot.KOM_IN.Profinet_PLC_INPUTS[3].6;														//30
	Robot.KOM_IN.Profinet_PLC_INPUTS[3].7;														//31

	//Vystupy z PLC do Robota//
	Robot.KOM_OUT.Profinet_PLC_OUTPUTS[0].0:= Robot.KOM_OUT.VypniMotory;						//0
	Robot.KOM_OUT.Profinet_PLC_OUTPUTS[0].1:= Robot.KOM_OUT.ZapniMotory;						//1
	Robot.KOM_OUT.Profinet_PLC_OUTPUTS[0].2:= Robot.KOM_OUT.PP_na_Main;							//2
	Robot.KOM_OUT.Profinet_PLC_OUTPUTS[0].3:= Robot.KOM_OUT.StartProgramu;						//3
	Robot.KOM_OUT.Profinet_PLC_OUTPUTS[0].4:= Robot.KOM_OUT.StartProgramuMain;					//4
	Robot.KOM_OUT.Profinet_PLC_OUTPUTS[0].5:= Robot.KOM_OUT.StopProgramu;						//5
	Robot.KOM_OUT.Profinet_PLC_OUTPUTS[0].6:= Robot.KOM_OUT.Reset_CS;							//6
	Robot.KOM_OUT.Profinet_PLC_OUTPUTS[0].7;													//7

	Robot.KOM_OUT.Profinet_PLC_OUTPUTS[1].0:= Robot.KOM_OUT.NalepEtiketu;						//8
	Robot.KOM_OUT.Profinet_PLC_OUTPUTS[1].1:= Robot.KOM_OUT.UkoncenieCykluRobota;				//9
	Robot.KOM_OUT.Profinet_PLC_OUTPUTS[1].2:= Robot.KOM_OUT.PresunDoMutingPozicie;				//10
	Robot.KOM_OUT.Profinet_PLC_OUTPUTS[1].3:= Robot.KOM_OUT.PresunDoPoziceKontrolyEtikety;		//11
	Robot.KOM_OUT.Profinet_PLC_OUTPUTS[1].4:= Robot.KOM_OUT.PresunDoPozicieKontrolyIntStitku;	//12
	Robot.KOM_OUT.Profinet_PLC_OUTPUTS[1].5:= Robot.KOM_OUT.PresunDoPozicieOdobratiaEtikety;	//13
	Robot.KOM_OUT.Profinet_PLC_OUTPUTS[1].6:= Robot.IN.PrisatieEtikety_OK_S1;					//14
	Robot.KOM_OUT.Profinet_PLC_OUTPUTS[1].7:= Robot.KOM_OUT.ServisnaPozicia;					//15

	Robot.KOM_OUT.Profinet_PLC_OUTPUTS[2].0:= Robot.KOM_OUT.ZahodEtiketu;						//16
	Robot.KOM_OUT.Profinet_PLC_OUTPUTS[2].1:= Robot.KOM_OUT.CitanieStitkuUkoncene; 				//17
	Robot.KOM_OUT.Profinet_PLC_OUTPUTS[2].2:= Robot.KOM_OUT.PresunDoPoziceKontrEtiketyPriamo;	//18
	Robot.KOM_OUT.Profinet_PLC_OUTPUTS[2].3;													//19
	Robot.KOM_OUT.Profinet_PLC_OUTPUTS[2].4;													//20
	Robot.KOM_OUT.Profinet_PLC_OUTPUTS[2].5;													//21
	Robot.KOM_OUT.Profinet_PLC_OUTPUTS[2].6;													//22
	Robot.KOM_OUT.Profinet_PLC_OUTPUTS[2].7;													//23

	Robot.KOM_OUT.Profinet_PLC_OUTPUTS[3].0:= Robot.KOM_OUT.LepenieStitku_ZnamienkoOffsetX;		//24
	Robot.KOM_OUT.Profinet_PLC_OUTPUTS[3].1:= Robot.KOM_OUT.LepenieStitku_ZnamienkoOffsetY;		//25
	Robot.KOM_OUT.Profinet_PLC_OUTPUTS[3].2:= Robot.KOM_OUT.LepenieStitku_ZnamienkoOffsetZ;		//26
	Robot.KOM_OUT.Profinet_PLC_OUTPUTS[3].3;													//27
	Robot.KOM_OUT.Profinet_PLC_OUTPUTS[3].4;													//28
	Robot.KOM_OUT.Profinet_PLC_OUTPUTS[3].5;													//29
	Robot.KOM_OUT.Profinet_PLC_OUTPUTS[3].6;													//30
	Robot.KOM_OUT.Profinet_PLC_OUTPUTS[3].7;													//31

	Robot.KOM_OUT.Profinet_PLC_OUTPUTS[4]:= Robot.KOM_OUT.CisloProduktu;						//32 - 39

	Robot.KOM_OUT.Profinet_PLC_OUTPUTS[5]:= Robot.KOM_OUT.LepenieStitku_OffsetX;				//40 - 47

	Robot.KOM_OUT.Profinet_PLC_OUTPUTS[6]:= Robot.KOM_OUT.LepenieStitku_OffsetY;				//48 - 55

	Robot.KOM_OUT.Profinet_PLC_OUTPUTS[7]:= Robot.KOM_OUT.LepenieStitku_OffsetZ;				//56 - 63

END_ACTION
```

#### KOM_Kamera.st
```iecst
ACTION KOM_Kamera:

	//Reset napájania kamery//
	IF Linka.ResetNapajaniaKamery THEN
		Linka.OUT.Rele_ResetNapajaniaKamery:= TRUE;
		Linka.ResetNapajaniaKamery:= FALSE;
	END_IF

	CasResetovaniaKamery.IN:= Linka.OUT.Rele_ResetNapajaniaKamery;
	IF CasResetovaniaKamery.Q THEN
		Linka.OUT.Rele_ResetNapajaniaKamery:= FALSE;
	END_IF

	CasResetovaniaKamery.PT:= T#2s;
	CasResetovaniaKamery();

	//Triger kamery//
	Kamera.Profinet_PLC_OUTPUTS.0:= Kamera.CMD.Triger;

	//Stav kamera READY//
	Kamera.STAV.READY:= StavHardware.Komunikacia_Kamera_OK;

	//Toogle bit kamery//
	Kamera.STAV.SWITCH:= Kamera.Profinet_PLC_INPUTS[4].0;

	//Stav - výsledky READY//
	IF EDGE(Kamera.STAV.SWITCH)THEN
		Kamera.STAV.Results_READY:= TRUE;
	END_IF

	//Stav - čítanie QR kódu alebi DM kódu OK//
	Kamera.RESULT.InternaEtiketa_QRkod_OK:= Kamera.Profinet_PLC_INPUTS[5].0;
	Kamera.RESULT.ZakazEtiketa_DMkod_OK:= Kamera.Profinet_PLC_INPUTS[5].1;
	Kamera.RESULT.ZakazEtiketa_PritomnZnakov_OK:= Kamera.Profinet_PLC_INPUTS[5].2;
	Kamera.RESULT.BielyPatern_OK:= Kamera.Profinet_PLC_INPUTS[5].3;

	//Vnútorné  počítadlo kamery//
	Kamera.STAV.RUN_Counter;

	//Zadané číslo programu kamery//
	Kamera.PAR.ZadaneCisloProgramu;

	//Číslo aktuálneho programu kamery//
	Kamera.STAV.AktualneCisloProgramu;

	//Zistenie počtu znakov Interného QR kódu//
	PocetNacitZnakovQRkodu := brsstrlen(ADR(Kamera.Profinet_InterEtiketaQRznaky));

	//Zistenie počtu znakov Zákaznického DM kódu//
	PocetNacitZnakovDMkodu := brsstrlen(ADR(Kamera.Profinet_ZakazEtiketaDMznaky));

	//Spájanie znakov Interného QR kódu z Pola USINT do výsledného stringu//
	brsmemcpy(ADR(Kamera.RESULT.InternaEtiketa_ZnakyQRkodu),ADR(Kamera.Profinet_InterEtiketaQRznaky),SIZEOF(Kamera.Profinet_InterEtiketaQRznaky));

	//Spájanie znakov Zákaznického DM kódu z Pola USINT do výsledného stringu//
	brsmemcpy(ADR(Kamera.RESULT.ZakazEtiketa_ZnakyDMkodu),ADR(Kamera.Profinet_ZakazEtiketaDMznaky),SIZEOF(Kamera.Profinet_ZakazEtiketaDMznaky));

END_ACTION
```

### Program Logical/Program/StoperDopravnikaNG (IEC)
